# B&R Automation Studio project TD52 (part 132)

### module_SA.typ - Package data types
```iecst
TYPE
	tVIS2MM : 	STRUCT
		bPI_SelfTest : BOOL; (* Switch port injection to selftest *) (* OldName:bSAFIPITest; Cycle: *)
		bCanUpDevSel : ARRAY[0..12]OF BOOL; (* CAN updater device selection *) (* OldName:new PV; Cycle: *)
		bCanUpStart : BOOL; (* CAN updater start/stop button *) (* OldName:new PV; Cycle: *)
		iCanUpFwVersSel : INT; (* CAN updater firmware version selection *) (* OldName:new PV; Cycle: *)
		bSAFI_SL_Check : BOOL; (* SAFI safty loop testing button *) (* OldName:bSAFI_SL_Check; Cycle: *)
		bSAFI_ValveLashSet : ARRAY[0..24]OF BOOL; (*Valve lash adjusted*)
		bSAFI_ValveLashSetAll : BOOL; (*Valve lash adjusted all*)
		bCanUpDevSelAll : BOOL; (*Update all button*)
	END_STRUCT;
	tMM2VIS : 	STRUCT
		iCnt_SA_ComErr : ARRAY[0..12]OF DINT; (* SAFI communication error counter *) (* OldName:usSAFIComErrCnt; Cycle:  *)
		iTi_PI_DurationAvg : INT; (* port injection duration average *) (* OldName:usDurationAvg; Cycle: *)
		iTi_PI_DurationMax : INT; (* port injection duration maximum *) (* OldName:usDurationMax; Cycle: *)
		iTi_PI_DurationMin : INT; (* port injection duration minimum *) (* OldName:usDurationMin; Cycle: *)
		tSA_HW_Vers : ARRAY[0..12]OF _tSAFIHardwareINT; (* SAFI hardware version *) (* OldName:usSAFIHW; Cycle: *)
		rSA_SW_Vers : ARRAY[0..12]OF REAL; (* SAFI software version *) (* OldName:usSAFIVers; Cycle: *)
		rTi_SA_OpHours : ARRAY[0..12]OF REAL; (* SAFI operating hours *) (* OldName:ulSAFArbH; Cycle: *)
		iSA_SerialNr : ARRAY[0..12]OF DINT; (* SAFI serial number *) (* OldName:ulSAFSerNr; Cycle: *)
		tSA_ProdDate : ARRAY[0..12]OF _tSAFIProdDateINT; (* SAFI production date *) (* OldName:ulProdDate; Cycle: *)
		rT_SA_ElecTemp : ARRAY[0..12]OF REAL; (* SAFI electronic temperature *) (* OldName:ssSAFITemp; Cycle: *)
		iSA_ErrToothNr : ARRAY[0..12]OF INT; (* SAFI Error tooth number *) (* OldName:usErrZahnz; Cycle: *)
		rSA_FiltVers : ARRAY[0..12]OF REAL; (* SAFI KLS filter version *) (* OldName:usSAFFiltV; Cycle: *)
		bMsg3337 : BOOL; (* Message number 3337 *) (* OldName:bACamSign; Cycle: *)
		bMsg3335 : BOOL; (* Message number 3335 *) (* OldName:bAOverspeedErr; Cycle: *)
		bMsg3333 : BOOL; (* Message number 3333 *) (* OldName:bAParameter; Cycle: *)
		bMsg2256 : BOOL; (* Message number 2256 *) (* OldName:bAPICloseErr; Cycle: *)
		bMsg2253 : BOOL; (* Message number 2253 (prepared V4.05.00*) (* OldName:Port injetion duration error; Cycle: *)
		bMsg2254 : BOOL; (* Message number 2254 *) (* OldName:bAPIHardwareErr; Cycle: *)
		bMsg2255 : BOOL; (* Message number 2255 *) (* OldName:bAPIOpenErr; Cycle: *)
		bMsg2281 : BOOL; (* Message number 2281 *) (* OldName:bAPBCMemBurst; Cycle: *)
		bMsg3331 : BOOL; (* Message number 3331 *) (* OldName:bASAFIComErr; Cycle: *)
		bMsg3336 : BOOL; (* Message number 3336 *) (* OldName:bATriggerSign; Cycle: *)
		bMsg3330 : BOOL; (* Message number 3330 *) (* OldName:bASAFIHwErr; Cycle: *)
		bMsg3332 : BOOL; (* Message number 3332 *) (* OldName:bASAFIWrongVers; Cycle: *)
		bMsg3334 : BOOL; (* Message number 3334 *) (* OldName:bAIPDeviation; Cycle: *)
		bMsg3338 : BOOL; (* Message number 3338 *) (* OldName:bAOutputErr; Cycle: *)
		bMsg3343 : BOOL; (* Message number 3343 *) (* OldName:bAMORISErr; Cycle: *)
		bMsg3344 : BOOL; (* Message number 3344 *) (* OldName:bIgnPowerFail; Cycle: *)
		bMsg3345 : BOOL; (* Message number 3345 *) (* OldName:bSAFISafetyLoop; Cycle: *)
		bMsg3277 : BOOL; (* Message number 3277 *) (* OldName:bBCamSign; Cycle: *)
		bMsg3292 : BOOL; (* Message number 3292 *) (* OldName:bBCanErrRate; Cycle: *)
		bMsg3291 : BOOL; (* Message number 3291 *) (* OldName:bBConfigErr; Cycle: *)
		bMsg3293 : BOOL; (* Message number 3293 *) (* OldName:bBElectrTemp; Cycle: *)
		bMsg3294 : BOOL; (* Message number 3294 *) (* OldName:bBIgnPwrLim; Cycle: *)
		bMsg2824 : BOOL; (* not used at the moment!? *) (* OldName:bBIGNShutOff; Cycle: *)
		bMsg3288 : BOOL; (* Message number 3288 *) (* OldName:bBIgnVoltMax; Cycle: *)
		bMsg3287 : BOOL; (* Message number 3287 *) (* OldName:bBIgnVoltMin; Cycle: *)
		bMsg3286 : BOOL; (* Message number 3286 *) (* OldName:bBOffsetErr; Cycle: *)
		bMsg3278 : BOOL; (* Message number 3278 *) (* OldName:bBOutputErr; Cycle: *)
		bMsg3275 : BOOL; (* Message number 3275 *) (* OldName:bBOverspeedErr; Cycle: *)
		bMsg3273 : BOOL; (* Message number 3273 *) (* OldName:bBParameter; Cycle: *)
		bMsg2820 : BOOL; (* not used at the moment!? *) (* OldName:bBPICloseErr; Cycle: *)
		bMsg2818 : BOOL; (* not used at the moment!? *) (* OldName:bBPIHardwareErr; Cycle: *)
		bMsg2819 : BOOL; (* not used at the moment!? *) (* OldName:bBPIOpenErr; Cycle: *)
		bMsg2823 : BOOL; (* not used at the moment!? *) (* OldName:bBPIShutOff; Cycle: *)
		bMsg3271 : BOOL; (* Message number 3271 cylinder info value *) (* OldName:bBSAFIComErr; Cycle: *)
		bMsg3276 : BOOL; (* Message number 3276 cylinder info value *) (* OldName:bBTriggerSign; Cycle: *)
		bMsg3270 : BOOL; (* Message number 3270 cylinder info value *) (* OldName:bBSAFIHwErr; Cycle: *)
		bMsg3283 : BOOL; (* Message number 3283 cylinder info value *) (* OldName:bBMORISErr; Cycle: *)
		bMsg3284 : BOOL; (* Message number 3284 cylinder info value *) (* OldName:bBSAFIFwErr; Cycle: *)
		bMsg3272 : BOOL; (* Message number 3272 cylinder info value *) (* OldName:bBSAFIWrongVers; Cycle: *)
		bMsg3274 : BOOL; (* Message number 3274 cylinder info value *) (* OldName:bBIPDeviation; Cycle: *)
		bMsg2816 : BOOL; (* Message number 2816 cylinder info value *) (* OldName:bPIOpen; Cycle: *)
		bMsg2817 : BOOL; (* Message number 2817 cylinder info value *) (* OldName:bPIOpen; Cycle: *)
		bMsg3536 : BOOL; (* Message number 3536 cylinder info value *) (* OldName:bWCamSign; Cycle: *)
		bMsg3531 : BOOL; (* Message number 3531 cylinder info value *) (* OldName:bWCanErrRate; Cycle: *)
		bMsg3535 : BOOL; (* Message number 3535 cylinder info value *) (* OldName:bWConfigErr; Cycle: *)
		bMsg3539 : BOOL; (* Message number 3539 cylinder info value *) (* OldName:bWElectrTemp; Cycle: *)
		bMsg3551 : BOOL; (* Message number 3551 cylinder info value *) (* OldName:bWIgnPwrLim; Cycle: *)
		bMsg3549 : BOOL; (* Message number 3549 cylinder info value *) (* OldName:bWIgnVoltAvg; Cycle: *)
		bMsg3550 : BOOL; (* Message number 3550 cylinder info value *) (* OldName:bWIgnVoltDev; Cycle: *)
		bMsg3548 : BOOL; (* Message number 3548 cylinder info value *) (* OldName:bWIgnVoltMax; Cycle: *)
		bMsg3547 : BOOL; (* Message number 3547 cylinder info value *) (* OldName:bWIgnVoltMin; Cycle: *)
		bMsg3546 : BOOL; (* Message number 3546 cylinder info value *) (* OldName:bWOffsetErr; Cycle: *)
		bMsg3545 : BOOL; (* Message number 3545 cylinder info value *) (* OldName:bWOutputErr; Cycle: *)
		bMsg2585 : BOOL; (* Message number 2585 cylinder info value *) (* OldName:bWPIHardwareErr; Cycle: *)
		bMsg3530 : BOOL; (* Message number 3530 cylinder info value *) (* OldName:bWSAFIComErr; Cycle: *)
		bMsg3537 : BOOL; (* Message number 3537 cylinder info value *) (* OldName:bWTriggerSign; Cycle: *)
		bMsg3533 : BOOL; (* Message number 3533 cylinder info value *) (* OldName:bWSAFIFwErr; Cycle: *)
		bMsg3544 : BOOL; (* Message number 3544 cylinder info value *) (* OldName:bWMORISErr; Cycle: *)
		iMsg3277 : INT; (* Message number 3277 cylinder info value *) (* OldName:ucCamSign; Cycle: *)
		iMsg3275 : INT; (* Message number 3275 cylinder info value *) (* OldName:ucOverspeedErr; Cycle: *)
		iMsg3273 : INT; (* Message number 3273 cylinder info value *) (* OldName:ucParameter; Cycle: *)
		iMsg2820 : INT; (* Message number 2820 cylinder info value *) (* OldName:ucPICloseErr; Cycle: *)
		iMsg2819 : INT; (* Message number 2819 cylinder info value *) (* OldName:ucPIOpenErr; Cycle: *)
		iMsg3271 : INT; (* Message number 3271 cylinder info value *) (* OldName:ucSAFIComErr; Cycle: *)
		iMsg3276 : INT; (* Message number 3276 cylinder info value *) (* OldName:ucTriggerSign; Cycle: *)
		iMsg3270 : INT; (* Message number 3270 cylinder info value *) (* OldName:ucSAFIHwErr; Cycle: *)
		iMsg3272 : INT; (* Message number 3272 cylinder info value *) (* OldName:ucSAFIWrongVers; Cycle: *)
		iMsg3274 : INT; (* Message number 3274 cylinder info value *) (* OldName:ucIPDeviation; Cycle: *)
		iMsg3278 : INT; (* Message number 3278 cylinder info value *) (* OldName:ucOutputErr; Cycle: *)
		iMsg3283 : INT; (* Message number 3283 cylinder info value *) (* OldName:ucMORISErr; Cycle: *)
		iMsg3292 : INT; (* Message number 3292 cylinder info value *) (* OldName:ucCanErrRate; Cycle: *)
		iMsg3291 : INT; (* Message number 3291 cylinder info value *) (* OldName:ucConfigErr; Cycle: *)
		iMsg3293 : INT; (* Message number 3293 cylinder info value *) (* OldName:ucElectrTemp; Cycle: *)
		iMsg3294 : INT; (* Message number 3294 cylinder info value *) (* OldName:ucIgnPwrLim; Cycle: *)
		iMsg3288 : INT; (* Message number 3288 cylinder info value *) (* OldName:ucIgnVoltMax; Cycle: *)
		iMsg3287 : INT; (* Message number 3287 cylinder info value *) (* OldName:ucIgnVoltMin; Cycle: *)
		iMsg3286 : INT; (* Message number 3286 cylinder info value *) (* OldName:ucOffsetErr; Cycle: *)
		iMsg2818 : INT; (* Message number 2818 cylinder info value *) (* OldName:ucPIHardwareErr; Cycle: *)
		iMsg3284 : INT; (* Message number 3284 cylinder info value *) (* OldName:ucSAFIFwErr; Cycle: *)
		bMsg3532 : BOOL; (* not used at the moment!? *) (* OldName:SAFI wrong type of software; Cycle: *)
		bMsg3534 : BOOL; (* not used at the moment!? *) (* OldName:SAFI  parameter failure; Cycle: *)
		bMsg3538 : BOOL; (* not used at the moment!? *) (* OldName:SAFI hardware failure; Cycle: *)
		bMsg3543 : BOOL; (* not used at the moment!? *) (* OldName:Ignition point deviation too high; Cycle: *)
		bMsg3552 : BOOL; (* SAFI ignition power module overload *) (* OldName:Ignition power supply overload; Cycle: *)
		bMsg3553 : BOOL; (* Message number 3553 *) (* OldName:bWPBCConfNotOK; Cycle: *)
		bMsg3554 : BOOL; (* Message number 3554 *) (* OldName:bWPBCInvalidPar; Cycle: *)
		bMsg2214 : BOOL; (* Message number 2214 *) (* OldName:bAPBCSigErr; Cycle: *)
		bMsg2297 : BOOL; (* PI correct current control rate message *) (* OldName:new PV; Cycle: *)
		bMsg2800 : BOOL; (* PI correct current control warning message *) (* OldName:new PV; Cycle: *)
		bMsg2906 : BOOL; (* PI correct current control warning message *) (* OldName:new PV; Cycle: *)
		iMsg2906 : INT; (* PI correct current control warning message *) (* OldName:new PV; Cycle: *)
		bMsg2298 : BOOL; (* PI demagnetisation failure message *) (* OldName:new PV; Cycle: *)
		bMsg2907 : BOOL; (* PI demagnetisation failure message *) (* OldName:new PV; Cycle: *)
		iMsg2907 : INT; (* PI demagnetisation failure message *) (* OldName:new PV; Cycle: *)
		iSA_ERZuV : ARRAY[0..24]OF INT; (* Error Rate for spark delay  *) (* OldName:ucERZuV; Cycle: *)
		iSA_ERDurTol : ARRAY[0..24]OF INT; (* Error Rate for Duration Tolerance  *) (* OldName:ucERDurTol; Cycle: *)
		rCanUpProgress : REAL; (* CAN updater progress bar *) (* OldName:new PV; Cycle: *)
		rCanUpFwVers : ARRAY[0..5]OF REAL; (* CAN updater firmware versions *) (* OldName:new PV; Cycle: *)
		bSAFI2 : BOOL; (* CAN updater SAFI2 detected *) (* OldName:new PV; Cycle: *)
		iSA_PICurGrad : ARRAY[0..24]OF INT; (* port injection close current gradient *) (* OldName:new PV; Cycle: *)
		iSA_PICurGradAvg : INT; (* port injection close current gradient average *) (* OldName:new PV; Cycle: *)
		iSA_PICurGradMax : INT; (* port injection close current gradient maximum *) (* OldName:new PV; Cycle: *)
		iSA_PICurGradMin : INT; (* port injection close current gradient minimum *) (* OldName:new PV; Cycle: *)
		bMsg2299 : BOOL; (* alarm A2299 cylinder pressure saturation replaced with warning W9318 if RKS enabled *) (* OldName:new PV; Cycle: *)
		bMsg9318 : BOOL; (* W9318 Cylinder pressure sensor saturation *) (* OldName:new PV; Cycle: *)
		bMsg2898 : BOOL; (* Message number 2898 cylinder info value *) (* OldName:new PV; Cycle: *)
		iMsg2898 : INT; (* Message number 2818 cylinder info value *) (* OldName:new PV; Cycle: *)
		bMsg2910 : BOOL; (* Message number 2910 cylinder info value *) (* OldName:new PV; Cycle: *)
		iMsg2910 : INT; (* Message number 2910 MPM info value *) (* OldName:new PV; Cycle: *)
		iMsg3344 : INT; (* Message number 3344 MPM  info value *) (* OldName:new PV; Cycle: *)
		iCMSmain_SAFI_status : INT; (* SAFI Module Main CMS Status *)
		iCMSinit_SAFI_status : INT; (* SAFI Module CMS Init Status *)
		bMsg2476 : BOOL; (*Message number 2476 SPAx CAM deviation monitoring*)
		iU_SAFI_Win3 : ARRAY[0..24]OF UINT; (*Outlet valve closure noise*)
		iU_SAFI_Win3_Min : UINT; (*Outlet valve closure noise min*)
		iU_SAFI_Win3_Max : UINT; (*Outlet valve closure noise max*)
		iU_SAFI_Win3_Avg : UINT; (*Outlet valve closure noise average*)
		iU_SAFI_Win4 : ARRAY[0..24]OF UINT; (*Inlet valve closure noise*)
		iU_SAFI_Win4_Min : UINT; (*Inlet valve closure noise min*)
		iU_SAFI_Win4_Max : UINT; (*Inlet valve closure noise max*)
		iU_SAFI_Win4_Avg : UINT; (*Inlet valve closure noise average*)
		iCA_SAFI_Win3 : ARRAY[0..24]OF UINT; (*Outlet valve closure timing*)
		iCA_SAFI_Win3_Min : UINT; (*Outlet valve closure timing min*)
		iCA_SAFI_Win3_Max : UINT; (*Outlet valve closure timing max*)
		iCA_SAFI_Win3_Avg : UINT; (*Outlet valve closure timing average*)
		iCA_SAFI_Win4 : ARRAY[0..24]OF UINT; (*Inlet valve closure timing*)
		iCA_SAFI_Win4_Min : UINT; (*Inlet valve closure timing min*)
		iCA_SAFI_Win4_Max : UINT; (*Inlet valve closure timing max*)
		iCA_SAFI_Win4_Avg : UINT; (*Inlet valve closure timing average*)
		bMsg2334 : BOOL; (*Alarm 2334 Outlet valve closure noise high*)
		bMsg9027 : BOOL; (*Operating message 9027 Outlet valve closure noise high*)
		iMsg9027 : UINT; (*Operating message 9027 Outlet valve closure noise high - Cylinder info*)
		bMsg2335 : BOOL; (*Alarm 2335 Outlet valve closure noise high*)
		bMsg9028 : BOOL; (*Operating message 9028 Outlet valve closure noise high*)
		iMsg9028 : UINT; (*Operating message 9028 Outlet valve closure noise high - Cylinder info*)
		bSA_VCD_Active : BOOL; (*Enable visualization of VCD parameters for legacy versions*)
		bMsg9320 : BOOL; (*Warning 9320 Exhaust valve unbalance*)
		bMsg9045 : BOOL; (*Operating message 9045 Exhaust valve unbalance*)
		iMsg9045 : UINT; (*Operating message 9045 Exhaust valve unbalance - Cylinder info*)
		bMsg9321 : BOOL; (*Warning 9321 Intake valve unbalance*)
		bMsg9046 : BOOL; (*Operating message 9046 Intake valve unbalance*)
		iMsg9046 : UINT; (*Operating message 9046 Intake valve unbalance - Cylinder info*)
		bMsg2493 : BOOL; (*Warning 2493 - SAFI measurements frozen or alternating*)
		bMsg2939 : BOOL; (*Operating message 2939 - SAFI measurements frozen or alternating*)
		iMsg2939 : UINT; (*Operating message 2939 - SAFI measurements frozen or alternating - Cylinder info*)
		bP_Red_SAErr_Bar : BOOL; (*Bit to activate the SAFI power reduction bar in the HMI*)
		bMsg9066 : BOOL; (*Operating message 9066 Cylinder pressure sensor measuring signal failure*)
		iMsg9066 : UINT; (*Operating message 9066 Cylinder pressure sensor measuring signal failure - Cylinder info*)
		bMsg9350 : BOOL; (*W9350 - KLS21 ignition monitoring not available*)
		bMsg9050 : BOOL; (*B9050 - KLS21 ignition monitoring not available*)
		iMsg9050 : UINT; (*B9050 - KLS21 ignition monitoring not available - cylinder number*)
		iNum_SafiType : ARRAY[0..12]OF USINT; (*Type of device. Unknown: 0. SAFI1: 1. SAFI2 KLS: 2. SAFI2 DMR: 3. SAFI3: 4. KLS21: 5.*)
		iNum_SafiUpdBlock : USINT; (*Block the CAN update procedure*)
		bSAFI3 : BOOL; (*All installed devices are not SAFI1*)
	END_STRUCT;
	_tSAFISpeed : 	STRUCT
		InCan : UINT;
		In : UINT;
		ValOK : UINT;
		Time : UDINT;
	END_STRUCT;
	_tSAFIProdDateINT : 	STRUCT
		YYYY : INT;
		MM : INT;
		DD : INT;
	END_STRUCT;
	_tSAFIProdDate : 	STRUCT
		YYYY : UINT;
		MM : USINT;
		DD : USINT;
	END_STRUCT;
	_tSAFICurrPmmREAL : 	STRUCT
		Current : REAL;
		Time : REAL;
	END_STRUCT;
	_tSAFICurrPmm : 	STRUCT
		Current : USINT;
		Time : UINT;
	END_STRUCT;
	_tSAFICurr : 	STRUCT
		Current_Low : USINT;
		Current_High : USINT;
		Time_Low : UINT;
		Time_High : UINT;
	END_STRUCT;
	_SAFIError : 	STRUCT
		Error : ARRAY[0..5]OF USINT;
	END_STRUCT;
	_tSAFImdatas : 	STRUCT
		data1 : UINT;
		data2 : UINT;
		data3 : UINT;
	END_STRUCT;
	_tSAFImdatasExtend : 	STRUCT
		data1 : UINT;
		data2 : UINT;
		data3 : UINT;
		data4 : USINT;
	END_STRUCT;
	_tSAFIHardwareINT : 	STRUCT
		HW_OPTION : INT;
		HW_VERSION : INT;
	END_STRUCT;
	_tSAFIHardware : 	STRUCT
		HW_OPTION : USINT;
		HW_VERSION : USINT;
	END_STRUCT;
	tE_SAFI : 	STRUCT
		Error : ARRAY[0..1]OF USINT;
		pdata : ARRAY[0..41]OF USINT;
		runstop : ARRAY[0..2]OF USINT;
		smdata : ARRAY[0..9]OF USINT;
	END_STRUCT;
	_tEventSAFI : 	STRUCT
		conf : ARRAY[0..35]OF USINT;
		zuend : ARRAY[0..1]OF USINT;
		error : USINT;
		sdata : ARRAY[0..4]OF USINT;
		idata : ARRAY[0..30]OF USINT;
		kdata : ARRAY[0..30]OF USINT;
		ddata : ARRAY[0..53]OF USINT;
		dmdata1 : ARRAY[0..5]OF USINT;
		kmdata : ARRAY[0..7]OF USINT;
		dmdata2 : ARRAY[0..15]OF USINT;
		smdata : ARRAY[0..9]OF USINT;
		status : ARRAY[0..11]OF USINT;
		bez : USINT;
		ref : USINT;
		cur : USINT;
		diag : ARRAY[0..18]OF USINT;
	END_STRUCT;
	tPIcurrentREAL : 	STRUCT
		current : REAL;
		duration : REAL;
	END_STRUCT;
	tPIrecoveryREAL : 	STRUCT
		delay : REAL;
		current : REAL;
		duration : REAL;
	END_STRUCT;
	tPIpulldet1REAL : 	STRUCT
		level : REAL;
		st_time : REAL;
	END_STRUCT;
	tPIopdet1REAL : 	STRUCT
		st_time : REAL;
		duration : REAL;
	END_STRUCT;
	tPIopdet2REAL : 	STRUCT
		grad_ul : REAL;
		grad_ll : REAL;
		rate : REAL;
	END_STRUCT;
	tPIclosdet1REAL : 	STRUCT
		set_current : REAL;
		set_duration : REAL;
	END_STRUCT;
	tPIclosdet2REAL : 	STRUCT
		duration : REAL;
		grad_curr : REAL;
		grad_curr_var : REAL;
	END_STRUCT;
	tPIaverageREAL : 	STRUCT
		average_MUX_6_7 : REAL;
		average_MUX_8_9 : REAL;
	END_STRUCT;
	CanDeviceGo : 	STRUCT
		CANDevGo : ARRAY[0..1]OF USINT;
		ECANDevGo : USINT;
	END_STRUCT;
	_tMonicLimitREAL : 	STRUCT
		limit : REAL;
		kind : REAL;
		delay : REAL;
	END_STRUCT;
	_tMonicLimit : 	STRUCT
		limit : USINT;
		kind : USINT;
		delay : USINT;
	END_STRUCT;
	IN_SA_struct : 	STRUCT
		iIdx_OMSS : INT; (* operationg mode selection switch *) (* OldName:BWS_HA; Cycle:5 *)
		iIdx_OMSS_TC2 : INT; (* operationg mode selection switch *) (* OldName:BWS_HA; Cycle:5 *)
		bEng_Dem_TC2 : BOOL; (* module demanded *) (* OldName:M_AGFD; Cycle:2 *)
		bEng_Dem : BOOL; (* module demanded *) (* OldName:M_AGFD; Cycle:5 *)
		iSt_OpMode : UDINT; (* engine operation mode *) (* OldName:StopM; Cycle:5 *)
		rCA_Ign_Act : ARRAY[0..24]OF REAL; (* actual cylinder ignition point *) (* OldName:ZZPCyl ; Cycle:2 *)
		bIgn_Dem_TC1 : BOOL; (* demand ignition *) (* OldName:ZUEND; Cycle:1 *)
		bIgn_Dem_TC2 : BOOL; (* demand ignition *) (* OldName:ZUEND; Cycle:2 *)
		bIgn_Dem : BOOL; (* demand ignition *) (* OldName:ZUEND; Cycle:5 *)
		bGV_On : BOOL; (* command open gas valves *) (* OldName:M_GASV; Cycle:2 *)
		tPIopenH : ARRAY[0..12]OF tPIopen; (* PI open point and open duration for high cylinder *) (* OldName:SAFI.tPI.tPIopenH; Cycle:2 *)
		tPIopenL : ARRAY[0..12]OF tPIopen; (* PI open point and open duration for low cylinder *) (* OldName:SAFI.tPI.tPIopenL; Cycle:2 *)
		bEng_Start_TC2 : BOOL; (*engine start*) (*OldName:M_STRT; Cycle:5*)
		bEng_Start : BOOL; (*engine start*) (*OldName:M_STRT; Cycle:5*)
		bIgn_SelfTest : BOOL; (* Switch ignition system to selftest  *) (* OldName:GoSelftest; Cycle:5 *)
		tAB2SA_TC2 : AmmBase2MM; (* AMM base to SAFI data transfer *) (* OldName:QUITT_WA; Cycle:2 *)
		tAB2SA : AmmBase2MM; (* AMM base to SAFI data transfer *) (* OldName:QUITT_WA; Cycle:5 *)
		iCANIdent : UDINT; (* CAN identifier from HalIO *) (* OldName:new PV; Cycle:7 *)
		iCANIdent_TC8 : UDINT; (* CAN identifier from HalIO *) (* OldName:new PV; Cycle:8 *)
		iCANIdentIGN2 : UDINT; (* CAN identifier of the 2nd CAN card from HalIO *) (* OldName:new PV; Cycle:8 *)
		iCANIdentIGN2_TC8 : UDINT; (* CAN identifier of the 2nd CAN card from HalIO *) (* OldName:new PV; Cycle:8 *)
		iMisfCyl : UDINT; (* cylinder misfire parameter *) (* OldName:MissfCyl; Cycle:2 *)
		iMisfCyl_TC2 : UDINT; (* cylinder misfire parameter *) (* OldName:MissfCyl; Cycle:2 *)
		tPB2MM : ParaBase2MM_type; (* Data exchange structure to ParaBase *) (* OldName:new PV; Cycle:5 *)
		tMO_PwrReply_TC5 : HALioDi_Type; (* DI: MORIS Ignition Power Module On *) (* OldName:DI_IgnPwrReply; Cycle:2 *)
		tMO_PwrReply : HALioDi_Type; (* DI: MORIS Ignition Power Module On *) (* OldName:DI_IgnPwrReply; Cycle:5 *)
		tMO_PwrReply2 : HALioDi_Type; (* DI: MORIS Ignition Power Module On *) (* OldName:new PV; Cycle:5 *)
		tMO_PwrReply3 : HALioDi_Type; (* DI: MORIS Ignition Power Module On *) (* OldName:new PV; Cycle:5 *)
		tMO_PwrReply4 : HALioDi_Type; (* DI: MORIS Ignition Power Module On *) (* OldName:new PV; Cycle:5 *)
		tMO_SaftyLoop_TC2 : HALioDi_Type; (* DI: MORIS Savety loop closed *) (* OldName:DI_MO_SL_OK; Cycle:2 *)
		tMO_SaftyLoop : HALioDi_Type; (* DI: MORIS Savety loop closed *) (* OldName:DI_MO_SL_OK; Cycle:5 *)
		tSafetyLoop_Eng_TC2 : HALioDi_Type; (* DI: Safety Loop closed *) (* OldName:RUHE; Cycle:2 *)
		tSafetyLoop_Eng : HALioDi_Type; (* DI: Safety Loop closed *) (* OldName:RUHE; Cycle:5 *)
		tMO_PowerOverload : HALioDi_Type; (* DI: SAFI ignition power module overload *) (* OldName:DI_IgnPowerOverload; Cycle:5 *)
		tMO_PowerOverload2 : HALioDi_Type; (* DI: SAFI ignition power module overload *) (* OldName:new PV; Cycle:5 *)
		tMO_PowerOverload3 : HALioDi_Type; (* DI: SAFI ignition power module overload *) (* OldName:new PV; Cycle:5 *)
		tMO_PowerOverload4 : HALioDi_Type; (* DI: SAFI ignition power module overload *) (* OldName:new PV; Cycle:5 *)
		tSafetyLoop_EmStop : HALioDi_Type; (* DI safety loop - emergency stop *) (* OldName:DI_SIS; Cycle:5 *)
		tGCB_On : HALioDi_Type; (*DI: generator circuit breaker closed *) (*OldName:GCB_ON; Cycle:2;*)
		tGCB_On_TC5 : HALioDi_Type; (*DI: generator circuit breaker closed *) (*OldName:GCB_ON; Cycle:2;*)
		iECanDevGo : USINT; (* event status CAN device go *) (* OldName:new PV; Cycle:2 *)
		bSimWinMOD_Active : BOOL; (* WinMode simulation active *) (* OldName:new PV; Cycle:2*)
		rP_Act_Norm_Filt : REAL; (* actual power related to rP_Nom filtered T=1s *) (*OldName:P_IST; Cycle:2*)
		rP_Act_Norm_Filt_TC5 : REAL; (* actual power related to rP_Nom filtered T=1s *) (*OldName:P_IST; Cycle:5*)
		iIdx_Gtyp_Dem : INT; (* actual gassort 1..4 *) (* OldName: gasart; Cycle:5; *)
		bLimpHomeCyl : ARRAY[0..24]OF BOOL; (* limp home if PBC in-cylinder pressure sensor failure *) (* OldName: bLimpHomeCyl; Cycle:2; *)
		bCUp_Man : ARRAY[0..24]OF BOOL; (* SAFI curve upload manuel selection *) (* OldName: ManualUpload; Cycle:2; *)
		rLam_Eng_LL_Set : REAL; (* Leanox Lambda set point *) (* OldName: ssPosGasmixerNominal; Cycle:2; *)
		rPr_Ch_P2s_Avg_TC2 : REAL; (* actual charge pressure before throttle valve (P2s) *) (* OldName: new PV; Cycle:2; *)
		rPr_Ch_P2s_Avg : REAL; (* actual charge pressure before throttle valve (P2s) *) (* OldName: new PV; Cycle:5; *)
		rT_Ch_T2s_Avg_TC2 : REAL; (* actual charge temperature (T2s) *) (* OldName: new PV; Cycle:2; *)
		rT_Ch_T2s_Avg : REAL; (* actual charge temperature (T2s) *) (* OldName: new PV; Cycle:5; *)
		bTrip_IPC_MSF : BOOL; (* Trip: A2214 Cylinder pressure sensor measuring signal failure Prio2*) (* OldName: bAKnockSigErr_DMR; Cycle:5; *)
		STP_STRT : BOOL; (*  tooth to tooth --> air starter off *) (* OldName: new PV; Cycle:5; *) (*V04.04.00.00*)
		bGridCode_ON : BOOL; (*any dyn. GridCode function activated*)
		bFastStart_ready_running : BOOL; (*Engine ready for fast start (engine stopped) OR fast start in action (until target load reached for the first time) *)
		bCANCntReset : BOOL; (* CAN error counter value reset *) (*OldName: bCANCounterReset; Cycle:5;*)
		tSPAx_CamDev : HALioDi_Type; (*DI: SPAx CAM deviation monitoring*) (* OldName: new PV; Cycle:5; *)
		bP_Red_SAErr : BOOL; (*Trigger SAFI power reduction*)
		bIC_IgnEngergy_Hi : BOOL; (*IC Warning Maximum Energy Exceeded*)
	END_STRUCT;
	OUT_SA_struct : 	STRUCT
		rN_IgnSAFI_Act : REAL; (* Engine speed measured by ignition SAFI *) (* OldName:ZDGSpeed; Cycle:2 *)
		bIgnOperating : BOOL; (* Ignition in Operation *) (* OldName:ZIB; Cycle:2 *)
		rT_EG_Cyl : ARRAY[0..24]OF REAL; (* cylinder exhaust gas temperatures *) (* OldName:t_zyl; Cycle:5 *)
		iU_SAFI_Win1 : ARRAY[0..24]OF INT; (* cylinder values of KLS window 1 *) (* OldName:Fenst1; Cycle:5 *)
		iU_SAFI_Win2 : ARRAY[0..24]OF INT; (* cylinder values of KLS window 2 *) (* OldName:Fenst2; Cycle:5 *)
		iU_SAFI_Win3 : ARRAY[0..24]OF INT; (* cylinder values of KLS window 3 *) (* OldName:Fenst3; Cycle:5 *)
		iU_SAFI_Win4 : ARRAY[0..24]OF INT; (* cylinder values of KLS window 4 *) (* OldName:Fenst4; Cycle:5 *)
		tMS_PBC0 : ARRAY[0..12]OF _tSAFImdatas; (* Pressure based control measuring data 0 *) (* OldName:DMR_md0; Cycle:5 *)
		tMS_PBC1 : ARRAY[0..12]OF _tSAFImdatas; (* Pressure based control measuring data 1 *) (* OldName:DMR_md1; Cycle:5 *)
		tMS_PBC2 : ARRAY[0..12]OF _tSAFImdatas; (* Pressure based control measuring data 2 *) (* OldName:DMR_md2; Cycle:5 *)
		tMS_PBC3 : ARRAY[0..12]OF _tSAFImdatas; (* Pressure based control measuring data 3 *) (* OldName:DMR_md3; Cycle:5 *)
		tMS_PBC4 : ARRAY[0..12]OF _tSAFImdatas; (* Pressure based control measuring data 4 *) (* OldName:DMR_md4; Cycle:5 *)
		tMS_PBC5 : ARRAY[0..12]OF _tSAFImdatas; (* Pressure based control measuring data 5 *) (* OldName:DMR_md5; Cycle:5 *)
		tMS_PBC6 : ARRAY[0..12]OF _tSAFImdatas; (* Pressure based control measuring data 6 *) (* OldName:DMR_md6; Cycle:5 *)
		tMS_PBC7 : ARRAY[0..12]OF _tSAFImdatas; (* Pressure based control measuring data 7 *) (* OldName:DMR_md7; Cycle:5 *)
		tMS_PBC8 : ARRAY[0..12]OF _tSAFImdatas; (* Pressure based control measuring data 8 *) (* OldName:DMR_md8; Cycle:5 *)
		tMS_PBC9 : ARRAY[0..12]OF _tSAFImdatas; (* Pressure based control measuring data 9 *) (* OldName:DMR_md9; Cycle:5 *)
		tMS_PBC10 : ARRAY[0..12]OF _tSAFImdatas; (* Pressure based control measuring data 10 *) (* OldName:DMR_md10; Cycle:5 *)
		tMS_PBC11 : ARRAY[0..12]OF _tSAFImdatas; (* Pressure based control measuring data 11 *) (* OldName:DMR_md11; Cycle:5 *)
		tMS_PBC12 : ARRAY[0..12]OF _tSAFImdatas; (* Pressure based control measuring data 12 *) (* OldName:DMR_md12; Cycle:5 *)
		tMS_PBC13 : ARRAY[0..12]OF _tSAFImdatas; (* Pressure based control measuring data 13 *) (* OldName:DMR_md13; Cycle:5 *)
		tMS_PBC14 : ARRAY[0..12]OF _tSAFImdatas; (* Pressure based control measuring data 14 *) (* OldName:DMR_md14; Cycle:5 *)
		tMS_PBC15 : ARRAY[0..12]OF _tSAFImdatas; (* Pressure based control measuring data 15 *) (* OldName:DMR_md15; Cycle:5 *)
		tMS_PBC16 : ARRAY[0..12]OF _tSAFImdatas; (* Pressure based control measuring data 16 *) (* OldName:DMR_md16; Cycle:5 *)
		tMS_PBC17 : ARRAY[0..12]OF _tSAFImdatas; (* Pressure based control measuring data 17 *) (* OldName:DMR_md17; Cycle:5 *)
		tMS_PBC18 : ARRAY[0..12]OF _tSAFImdatas; (* Pressure based control measuring data 18 *) (* OldName:DMR_md18; Cycle:5 *)
		tMS_PBC19 : ARRAY[0..12]OF _tSAFImdatas; (* Pressure based control measuring data 19 *) (* OldName:DMR_md19; Cycle:5 *)
		tMS_PBC20 : ARRAY[0..12]OF _tSAFImdatasExtend; (* Pressure based control measuring data 20*)
		tMS_PBC21 : ARRAY[0..12]OF _tSAFImdatasExtend; (* Pressure based control measuring data 21*)
		b_IgnSAFI_SelfTestBack : BOOL; (* Feedback: Ignition system SAFI is in selftest mode *) (* OldName:bSAFISelfTest; Cycle:5 *)
		rU_IgnSAFI_Max : REAL; (* maximum ignition voltage  *) (* OldName:MaxVolt; Cycle:5 *)
		rU_IgnSAFI_Min : REAL; (* minimum ignition voltage  *) (* OldName:MinVolt; Cycle:5 *)
		rU_IgnSAFI_Cyl : ARRAY[0..24]OF REAL; (* ignition voltage for each cylinder  *) (* OldName:V_Zyl; Cycle:5 *)
		rU_IgnSAFI_Avg : REAL; (* ignition voltage average *) (* OldName:AvgVolt; Cycle:5 *)
		tSAFI_CanGo : CanDeviceGo; (* Start / Stop CAN communication *) (* OldName:CANDevGo; Cycle:5 *)
		rN_IgnSAFI_LastValOK : REAL; (* last sent speed value from one of the SAFI devices *) (* OldName:n_lastValOK; Cycle:2 *)
		tSA2AB : MM2AmmBase; (* SAFI module to AMM base data transfer *) (* OldName:new PV; Cycle:2 *)
		tSA2PB : MM2ParaBase_type; (* Data exchange structure to ParaBase *) (* OldName:new PV; Cycle:5 *)
		tMO_PwrRequest : HALioDo_Type; (* DO: MORIS Ignition Power Module Request *) (* OldName:DO_IgnPwrRequest; Cycle:5 *)
		tMO_PwrRequest2 : HALioDo_Type; (* DO: MORIS Ignition Power Module Request *) (* OldName:new PV; Cycle:5 *)
		tMO_PwrRequest3 : HALioDo_Type; (* DO: MORIS Ignition Power Module Request *) (* OldName:new PV; Cycle:5 *)
		tMO_PwrRequest4 : HALioDo_Type; (* DO: MORIS Ignition Power Module Request *) (* OldName:new PV; Cycle:5 *)
		bPBCSensErr : ARRAY[0..24]OF BOOL; (* error info for PBC *) (* OldName:bZM_PBCSensErr; Cycle:5 *)
		bPBCCompLineCheck : ARRAY[0..24]OF BOOL; (* error info for PBC *) (* OldName:bPBCCompLineCheck; Cycle:5 *)
		bPBCNegVoltCheck : ARRAY[0..24]OF BOOL; (* error info for PBC *) (* OldName:bPBCNegVoltCheck; Cycle:5 *)
		bPBCNegPresCheck : ARRAY[0..24]OF BOOL; (* error info for PBC *) (* OldName:bPBCNegPresCheck; Cycle:5 *)
		bPBCPresSlopeCheck : ARRAY[0..24]OF BOOL; (* error info for PBC *) (* OldName:bPBCPresSlopeCheck; Cycle:5 *)
		bPBCSlowDriftCheck : ARRAY[0..24]OF BOOL; (* error info for PBC *) (* OldName:bPBCSlowDriftCheck; Cycle:5 *)
		bPBCConfNotOK : ARRAY[0..12]OF BOOL; (* error info for PBC *) (* OldName:bPBCConfNotOK; Cycle:5 *)
		bPBCMemBurst : ARRAY[0..24]OF BOOL; (* error info for PBC *) (* OldName:bPBCMemBurst; Cycle:5 *)
		bSAFIPBCConfNotOK : BOOL; (* blocking of start because SAFI PBC parameter are not valid *) (* OldName:bSAFIPBCConfNotOK; Cycle:2 *)
		tCUp : ARRAY[0..24]OF tCup_Perm; (* SAFI curve upload data *) (* OldName:tCup; Cycle:2 *)
		iCUpStack : ARRAY[0..23]OF USINT; (* SAFI curve upload stack *) (* OldName:Stack; Cycle:2 *)
		bPBCInvalidPar : ARRAY[0..12]OF BOOL; (* SAFI invalid PBC parameter *) (* OldName:bPBCInvalidPar; Cycle:2 *)
		rSA_SW_Vers : ARRAY[0..12]OF REAL; (* SAFI software version *) (* OldName:usSAFIVers; Cycle: *)
		rSA_FiltVers : ARRAY[0..12]OF REAL; (* SAFI KLS filter version *) (* OldName:usSAFFiltV; Cycle: *)
		rT_SA_ElecTemp : ARRAY[0..12]OF REAL; (* SAFI electronic temperature *) (* OldName:ssSAFITemp; Cycle: *)
		rSA_PBC_Sens : ARRAY[0..12]OF REAL; (* PBC sensor sensitivity [mV/bar] *) (* new PV; Cycle: 2*)
		bPBCCPSSat : ARRAY[0..24]OF BOOL; (* Cylinder pressure sensor saturation flag for cyl X *) (* new PV; Cycle: 2*)
		tE_SAFI : ARRAY[0..12]OF _tEventSAFI; (* SAFI CAN Events *)
		iCnt_SA_ComErr : ARRAY[0..12]OF DINT; (* SAFI communication error counter *) (* OldName:usSAFIComErrCnt; Cycle:  *)
		iSA_ERZuV : ARRAY[0..24]OF INT; (* Error Rate for spark delay  *) (* OldName:ucERZuV; Cycle: *)
		iSA_ERDurTol : ARRAY[0..24]OF INT; (* Error Rate for Duration Tolerance  *) (* OldName:ucERDurTol; Cycle: *)
		bSA_PBCFrozenAltern : ARRAY[0..24]OF BOOL; (*DMR knock signal or IMEP frozen or alternating*)
		bSA_Win1FrozenAltern : ARRAY[0..24]OF BOOL; (*Knock noise signal frozen or alternating*)
		iT_EG_CylFault : ARRAY[0..24]OF UINT; (*0 = No fault / bit0 = SAFI re-para active / bit1 = Exhaust gas temperature signal frozen or alternating*)
		rP_Red_SAErr_Norm : REAL; (* Power reduction by CAN communication failure for half or more SAFI or too many SAFI reboots*)
		bSA_CfgDone : BOOL; (*All SAFI in operation mode*)
		rIHR : ARRAY[0..24]OF REAL; (*Integrated heat release [kJ/m2]*)
		rU_Ign_Max_LimHi : REAL; (* Maximum ignition voltage high limit *)
		bMsg9318_Set : BOOL; (* W9318 cylinder pressure sensor saturation is set *)
	END_STRUCT;
	tPIclosgrad : 	STRUCT
		PICurGrad : INT;
		PCICurGrad : INT;
	END_STRUCT;
	tPIMode : 	STRUCT
		EnabRun : BOOL;
		PIself : BOOL;
		PCIself : BOOL;
		PIclose : BOOL;
		PCIclose : BOOL;
		MAct_6_7 : BOOL;
		MAct_8_9 : BOOL;
		Bit08 : BOOL;
		Bit09 : BOOL;
		Bit10 : BOOL;
		Bit11 : BOOL;
		Bit12 : BOOL;
		Bit13 : BOOL;
		Bit14 : BOOL;
		Bit15 : BOOL;
		Bit16 : BOOL;
	END_STRUCT;
	tPIopen : 	STRUCT
		timing : UINT;
		duration : UINT;
	END_STRUCT;
	tPIcurrent : 	STRUCT
		current : USINT;
		duration : UINT;
	END_STRUCT;
	tPIrecovery : 	STRUCT
		delay : UINT;
		current : SINT;
		duration : UINT;
	END_STRUCT;
	tPIaverage : 	STRUCT
		average_MUX_6_7 : USINT;
		average_MUX_8_9 : USINT;
	END_STRUCT;
	tPICurGrad : 	STRUCT
		ssFiFo : ARRAY[0..10]OF INT;
		slSum : DINT;
		ssAvg : INT;
	END_STRUCT;
	tPI : 	STRUCT
		Mode : UINT;
		tPIopenH : tPIopen;
		tPIopenL : tPIopen;
		tPIcurr1 : tPIcurrent;
		tPIcurr2 : tPIcurrent;
		tPIcurr3 : tPIcurrent;
		PIcurr4 : USINT;
		tPIrecov : tPIrecovery;
		tPIpudet1 : tPIpulldet1;
		tPIpudet2 : tPIpulldet2;
		tPIpudet3 : tPIpulldet3;
		tPIopdet1 : tPIopdet1;
		tPIopdet2 : tPIopdet2;
		tPIopdet3 : tPIopdet3;
		tPIopdet4 : tPIopdet4;
		PIclotim : UINT;
		tPIclodet0 : tPIclosdet0;
		tPIclodet1 : tPIclosdet1;
		tPIclodet2 : tPIclosdet2;
		tPIclodet3 : tPIclosdet3;
		tPIclodet4 : tPIclosdet4;
		tPIclodet5 : tPIclosdet5;
		tPCopenH : tPCopen;
		tPCopenL : tPCopen;
		tPCcurr1 : tPCcurrent;
		tPCcurr2 : tPCcurrent;
		tPCcurr3 : tPCcurrent;
		PCcurr4 : USINT;
		tPCrecov : tPCrecovery;
		tPCpudet1 : tPCpulldet1;
		tPCpudet2 : tPCpulldet2;
		tPCopdet1 : tPCopdet1;
		tPCopdet2 : tPCopdet2;
		tPCopdet3 : tPCopdet3;
		tPCfree : tPCfree;
		PCclodet1 : UINT;
		tPCclodet2 : tPCclosdet2;
		tPCclodet3 : tPCclosdet3;
		ShOffRate : USINT;
		tAverage : tPIaverage;
		tPIdemagL : tPIdemag;
		tPIdemagH : tPIdemag;
		tPIcurrCtrL : tPIcurrCtrL;
		tPIcurrCtrH : tPIcurrCtrH;
		ucValveON : USINT;
		tVaOpenL : _tSAFImdatas;
		tVaOpenH : _tSAFImdatas;
		tCurrGradL : tPIclosgrad;
		tCurrGradH : tPIclosgrad;
	END_STRUCT;
	tSAFI : 	STRUCT
		tPI : tPI;
		tError : ARRAY[0..1]OF _SAFIError;
		E_SAFI : tE_SAFI;
	END_STRUCT;
	tPIpulldet1 : 	STRUCT
		level_L : UINT;
		level_H : UINT;
	END_STRUCT;
	tPIpulldet2 : 	STRUCT
		st_time_L : UINT;
		st_time_H : UINT;
	END_STRUCT;
	tPIpulldet3 : 	STRUCT
		duration_L : UINT;
		duration_H : UINT;
		rate : USINT;
	END_STRUCT;
	tPIopdet1 : 	STRUCT
		st_time_L : UINT;
		st_time_H : UINT;
	END_STRUCT;
	tPIopdet2 : 	STRUCT
		duration_L : UINT;
		duration_H : UINT;
	END_STRUCT;
	tPIopdet3 : 	STRUCT
		up_level_L : UINT;
		up_level_H : UINT;
	END_STRUCT;
	tPIopdet4 : 	STRUCT
		lo_level_L : UINT;
		lo_level_H : UINT;
		rate : USINT;
	END_STRUCT;
	tPIclosdet0 : 	STRUCT
		FailR_L : UINT;
		FailR_H : UINT;
	END_STRUCT;
	tPIclosdet1 : 	STRUCT
		st_time_L : UINT;
		st_time_H : UINT;
	END_STRUCT;
	tPIclosdet2 : 	STRUCT
		set_current_L : USINT;
		set_current_H : USINT;
	END_STRUCT;
	tPIclosdet3 : 	STRUCT
		set_duration_L : UINT;
		set_duration_H : UINT;
	END_STRUCT;
	tPIclosdet4 : 	STRUCT
		duration_L : UINT;
		duration_H : UINT;
		cur_gradient_L : INT;
	END_STRUCT;
	tPIclosdet5 : 	STRUCT
		cur_gradient_H : INT;
		var_limit_L : UINT;
		var_limit_H : UINT;
	END_STRUCT;
	tPCopen : 	STRUCT
		timing : UINT;
		duration : UINT;
	END_STRUCT;
	tPCcurrent : 	STRUCT
		current : USINT;
		duration : UINT;
	END_STRUCT;
	tPCrecovery : 	STRUCT
		delay : UINT;
		current : SINT;
		duration : UINT;
	END_STRUCT;
	tPCpulldet1 : 	STRUCT
		level : UINT;
		st_time : UINT;
	END_STRUCT;
	tPCpulldet2 : 	STRUCT
		duration : UINT;
		current : UINT;
		rate : USINT;
	END_STRUCT;
	tPCopdet1 : 	STRUCT
		st_time : UINT;
		duration : UINT;
	END_STRUCT;
	tPCopdet2 : 	STRUCT
		upper_lvl : UINT;
		lower_lvl : UINT;
		rate : USINT;
	END_STRUCT;
	tPCopdet3 : 	STRUCT
		min_curr : UINT;
		rate : USINT;
	END_STRUCT;
	tPCfree : 	STRUCT
		free : UINT;
	END_STRUCT;
	tPCclosdet2 : 	STRUCT
		set_current : USINT;
		set_duration : UINT;
	END_STRUCT;
	tPCclosdet3 : 	STRUCT
		duration : UINT;
		grad_curr : INT;
		grad_curr_var : UINT;
	END_STRUCT;
	tDMR_ref : 	STRUCT
		boost_pr : INT;
		mix_temp : INT;
	END_STRUCT;
	Pressure : 	STRUCT
		Low : ARRAY[0..719]OF UINT;
		LowCA : ARRAY[0..719]OF UINT;
		High : ARRAY[0..719]OF UINT;
		HighCA : ARRAY[0..719]OF UINT;
	END_STRUCT;
	tCup_Pm : 	STRUCT
		Perm : ARRAY[0..24]OF tCup_Perm;
	END_STRUCT;
	tCup_Perm : 	STRUCT
		Press : ARRAY[0..719]OF UINT;
		day : UINT;
		month : UINT;
		year : UINT;
		hour : UINT;
		minute : UINT;
		millisec : UDINT;
		rLam_Eng_LL_Set : REAL;
		rPr_Eng_P2s : REAL;
		rT_Eng_T2s : REAL;
		rP_Act_Norm_Filt : REAL;
	END_STRUCT;
	rtctime_typ : 	STRUCT
		year : UINT;
		month : USINT;
		day : USINT;
		reserve : USINT;
		hour : USINT;
		minute : USINT;
		second : USINT;
		millisec : UINT;
		microsec : UINT;
	END_STRUCT;
	tPIdemag : 	STRUCT
		delay : UINT;
		duration : UINT;
		up_limit : USINT;
	END_STRUCT;
	tPIcurrCtrL : 	STRUCT
		delay : UINT;
		duration : UINT;
		level : USINT;
	END_STRUCT;
	tPIcurrCtrH : 	STRUCT
		delay : UINT;
		duration : UINT;
		level : USINT;
		rate : USINT;
	END_STRUCT;
	tDiag : 	STRUCT
		ParaFail : tParaFail;
	END_STRUCT;
	tParaFail : 	STRUCT
		Id : UINT;
		Mux : USINT;
		Nr : USINT;
	END_STRUCT;
END_TYPE
```

### Module_SAPara.typ - Package data types
```iecst
TYPE
	PROGRAMMER_INFO : 	STRUCT
		DO_NOT_SORT_PARA : STRING[40] := 'DO NOT CHANGE PARAMETER SORTING!'; (*DO NOT CHANGE PARAMETER SORTING!*) (*ADD NEW PARAMETER ONLY AT THE END OF THE Para STRUCTURE. DO NOT DELETE existing Para items.*)
	END_STRUCT;
	Para_SA_struct : 	STRUCT
		rCA_AdvTimeLim : REAL; (*PARA [12065]: advanced ingnition timing 1/10 deg *) (* OldName:AdvTimLi; Cycle: *)
		bSA_PI_CloDetActive : BOOL; (*PARA [12121]: TRUE = SAFI PI close detection is enabled/active *) (* OldName:bCloDet_Act; Cycle: *)
		bSA_Active : BOOL; (*PARA [12114]: TRUE = SAFI is enabled/active *) (* OldName:bSAFI_Act; Cycle: *)
		bSA_PBC_Active : BOOL; (*PARA [12119]: TRUE = SAFI PBC function is enabled/active *) (* OldName:bSAFIDMR_Act; Cycle: *)
		bSA_EG_Active : BOOL; (*PARA [12115]: TRUE = SAFI exh. temp. measur. is enabled/active *) (* OldName:bSAFIExhT_Act; Cycle: *)
		bSA_HV_Active : BOOL; (*PARA [12116]: TRUE = SAFI high volt. measur. is enabled/active *) (* OldName:bSAFIHS_Act; Cycle: *)
		bSA_Ign_Active : BOOL; (*PARA [12117]: TRUE = SAFI ignition function is enabled/active *) (* OldName:bSAFIIgn_Act; Cycle: *)
		bSA_KLS_Active : BOOL; (*PARA [12118]: TRUE = SAFI KLS function is enabled/active *) (* OldName:bSAFIKLS_Act; Cycle: *)
		bSA_PI_Active : BOOL; (*PARA [12120]: TRUE = SAFI port injection is enabled/active *) (* OldName:bSAFIPI_Act; Cycle: *)
		rN_EngNom : REAL; (*PARA [12128]: engine nominal speed *) (* OldName:n_nenn; Cycle: *)
		rN_OvrSpeed : REAL; (*PARA [12129]: Ignition overspeed limit *) (* OldName:OvrSpeed; Cycle: *)
		rCA_RetTimeLim : REAL; (*PARA [12066]: Retard ignition timing limit 1/10 deg  *) (* OldName:RetTimLi; Cycle: *)
		rSA_PI_opdet2_rate : REAL; (*PARA [12145]: SAFI PI opdet2_rate *) (* OldName:SAFI_tPI_tPIopdet2_ratePMM; Cycle: *)
		rSA_PI_pudet2_rate : REAL; (*PARA [12146]: SAFI PI pudet2_rate *) (* OldName:SAFI_tPI_tPIpudet2_ratePMM; Cycle: *)
		tSA_Ign_0 : _tSAFICurrPmmREAL; (* Para: SAFI ignition current / duration setting 0 *) (* OldName:SAFICurr0PMM; Cycle: *)
		tSA_Ign_1 : _tSAFICurrPmmREAL; (* Para: SAFI ignition current / duration setting 1 *) (* OldName:SAFICurr1PMM; Cycle: *)
		tSA_Ign_2 : _tSAFICurrPmmREAL; (* Para: SAFI ignition current / duration setting 2 *) (* OldName:SAFICurr2PMM; Cycle: *)
		tSA_Ign_3 : _tSAFICurrPmmREAL; (* Para: SAFI ignition current / duration setting 3 *) (* OldName:SAFICurr3PMM; Cycle: *)
		tSA_Ign_4 : _tSAFICurrPmmREAL; (* Para: SAFI ignition current / duration setting 4 *) (* OldName:SAFICurr4PMM; Cycle: *)
		tSA_Ign_5 : _tSAFICurrPmmREAL; (* Para: SAFI ignition current / duration setting 5 *) (* OldName:SAFICurr5PMM; Cycle: *)
		tSA_Ign_6 : _tSAFICurrPmmREAL; (* Para: SAFI ignition current / duration setting 6 *) (* OldName:SAFICurr6PMM; Cycle: *)
		rSA_PBC_Sensitivity : REAL; (*PARA [12144]: PBC sensor sensitivity [mV/bar] *) (* OldName:ssDMR_empf; Cycle: *)
		rSA_ResetPos : REAL; (*PARA [12148]: SAFI reset position *) (* OldName:ssPosResSA; Cycle: *)
		rSA_EarlTiIonization : REAL; (*PARA [12135]: earliest timing for ionization *) (* OldName:ucAdvTiIonPMM; Cycle: *)
		rSA_CoilType : REAL; (*PARA [12130]: coil type *) (* OldName:ucCoilType; Cycle: *)
		rSA_DelFailR : REAL; (*PARA [12131]: trip limit spark delay failure rate *) (* OldName:ucDelFailRPMM; Cycle: *)
		rSA_DeMagLvl : REAL; (*PARA [12132]: magnatism level decrease *) (* OldName:ucDeMagLvlPMM; Cycle: *)
		rSA_DurFailR : REAL; (*PARA [12133]: spark duration deviation failure rate *) (* OldName:ucDurFailR; Cycle: *)
		rSA_DurTol : REAL; (*PARA [12134]: spark duration deviation limit *) (* OldName:ucDurTol; Cycle: *)
		rSA_InMagLvl : REAL; (*PARA [12140]: magnatism level increase *) (* OldName:ucInMagLvlPmm; Cycle: *)
		rSA_MxSpPow : REAL; (*PARA [12143]: limit for spark power *) (* OldName:ucMxSpPowPMM; Cycle: *)
		iSA_PIValveType : INT; (*PARA [12147]: valve type (1=Woodward, 2= Hoerbiger)*) (* OldName:ucPIValveType; Cycle: *)
		rSA_RetTiIon : REAL; (*PARA [12149]: latest timing for ionization *) (* OldName:ucRetTiIonPMM; Cycle: *)
		rSA_SparkCurChar : REAL; (*PARA [12150]: spark current characteristic *) (* OldName:ucSparkCurChar; Cycle: *)
		rSA_SparkCurLev : REAL; (*PARA [12151]: spark current level *) (* OldName:ucSparkCurLev; Cycle: *)
		rSA_SpPOffTi : REAL; (*PARA [12153]: turn on/off ration for spark power *) (* OldName:ucSpPOffTiPMM; Cycle: *)
		rSA_SparkDuration : REAL; (*PARA [12152]: SAFI spark duration  *) (* OldName:usDurationPMM; Cycle: *)
		rSA_Eps : REAL; (*PARA [12136]: eps *) (* OldName:usEps; Cycle: *)
		rSA_IgnPwrLi : REAL; (*PARA [12138]: SAFI ignition  power limitation  *) (* OldName:usIgnPwrLi; Cycle: *)
		rSA_IgnPwrOut : REAL; (*PARA [12139]: power supply output *) (* OldName:usIgnPwrOut; Cycle: *)
		rSA_MxIonMag : REAL; (*PARA [12141]: magnatism ionisation level *) (* OldName:usMxIonMagPMM; Cycle: *)
		rSA_MxMagLvl : REAL; (*PARA [12142]: magnatism level limit *) (* OldName:usMxMagLvlPMM; Cycle: *)
		rSA_IgnFeedbackLim : REAL; (*PARA [12137]: Time for ignition feedback *) (* OldName:usZuVLimPMM; Cycle: *)
		rCA_Win1_B : REAL; (*PARA [12122]: beginn of window 1 in 1/10 deg.  *) (* OldName:WMF1_B; Cycle: *)
		rCA_Win1_D : REAL; (*PARA [12123]: duration of window 1 in 1/10 deg.  *) (* OldName:WMF1_D; Cycle: *)
		rCA_Win2_B : REAL; (*PARA [12124]: beginn of window 2 in 1/10 deg.  *) (* OldName:WMF2_B; Cycle: *)
		rCA_Win2_D : REAL; (*PARA [12125]: duration of window 2 in 1/10 deg.  *) (* OldName:WMF2_D; Cycle: *)
		rCA_Win3_B : REAL; (*PARA [12126]: beginn of window 3 in 1/10 deg.  *) (* OldName:WMF3_B; Cycle: *)
		rCA_Win3_D : REAL; (*PARA [12127]: duration of window 3 in 1/10 deg.  *) (* OldName:WMF3_D; Cycle: *)
		rCA_Win4_B : REAL; (*PARA [14310]: beginn of window 4 in 1/10 deg.  *) (* OldName:WMF4_B; Cycle: *)
		rCA_Win4_D : REAL; (*PARA [14311]: duration of window 4 in 1/10 deg.  *) (* OldName:WMF4_D; Cycle: *)
		rSA_Win1_F : REAL; (*PARA [12154]: window 1 function *) (* OldName:FenstF1; Cycle: *)
		rSA_Win2_F : REAL; (*PARA [14312]: window 2 function *) (* OldName:FenstF2; Cycle: *)
		rSA_Win3_F : REAL; (*PARA [14313]: window 3 function *) (* OldName:FenstF3; Cycle: *)
		rSA_Win4_F : REAL; (*PARA [14314]: window 4 function *) (* OldName:FenstF4; Cycle: *)
		rU_IgnMon_LimActive : REAL; (*PARA [12155]: ignition voltage start monitoring  *) (* OldName:LimitActiv; Cycle: *)
		tIgn_LimitMonitor : ARRAY[0..4]OF _tMonicLimitREAL; (* Para: parameter voltage limit monitoring  *) (* OldName:LimitMon; Cycle: *)
		bIgn_LimitMonitorActive : ARRAY[0..4]OF BOOL; (* Para: type of voltage limit monitoring *) (* OldName:MonLimitOn; Cycle: *)
		bGridCode_Active : BOOL; (*PARA [11055]: Gride Code active *) (* OldName:bGridCode; Cycle: *)
		iEng_Motortype : INT; (* Para: Engine type *) (* OldName:motortyp; Cycle: *)
		bGridCodeMonitoringOnly : BOOL; (*PARA [11056]: Grid Code monitoring only active *) (* OldName:bGridCodeMonitoringOnly; Cycle: *)
		zz_V4_0_ParaVersionEnd : REAL := 4.0; (*! ADD NEW PARAMETER ONLY BELOW THIS LINE ! This is the end of base version parameter and has to stay unchanged. DO NOT CHANGE SORT ORDER of Para!*) (* OldName: new PV; Cycle: 5; *)
		rHCR : ARRAY[0..4]OF REAL; (* Para: Heat Capacity Ratio *) (* OldName: rKappa; Cycle: 2 *)
		bGT_SpecGasActive : BOOL; (*PARA [11374]: Sondergas *)
		bDynSparkDuration : BOOL; (*PARA [13646]: Variable spark duration active *) (* OldName:newPV; Cycle: *)
		usDurationIdle : UINT; (*PARA [13647]: Spark duration below power threshold *) (* OldName:newPV; Cycle: *)
		rP_Act_DynSpark_Limit_Nom : REAL; (*PARA [13648]: Spark duration below power threshold *) (* OldName:newPV; Cycle: *)
		iSA_CyclPIOnDuringMisf : USINT; (*PARA [13698]: Allowed Nr of cycles of ign off with PI on during misfire*) (* OldName:newPV; Cycle: *)
		rSA_PI_pudet_level : REAL; (*PARA [13699]: PI pull in current level *) (* OldName:newPV; Cycle: *)
		rSA_PI_pudet_st_time : REAL; (*PARA [13700]: PI pull in current start time *) (* OldName:newPV; Cycle: *)
		rSA_PI_pudet_duration : REAL; (*PARA [13701]: PI pull in current duration *) (* OldName:newPV; Cycle: *)
		rSA_PI_demag_delay : REAL; (*PARA [13707]: PI demagnetisation delay *) (* OldName:newPV; Cycle: *)
		rSA_PI_demag_duration : REAL; (*PARA [13708]: PI demagnetisation duration  *) (* OldName:newPV; Cycle: *)
		rSA_PI_demag_up_limit : REAL; (*PARA [13709]: PI demagnetisation upper limit *) (* OldName:newPV; Cycle: *)
		rSA_PI_currCtr_delay : REAL; (*PARA [13702]: PI correct current control delay *) (* OldName:newPV; Cycle: *)
		rSA_PI_currCtr_duration : REAL; (*PARA [13703]: PI correct current control duration *) (* OldName:newPV; Cycle: *)
		rSA_PI_currCtr_level : REAL; (*PARA [13704]: PI correct current control level *) (* OldName:newPV; Cycle: *)
		rSA_PI_currCtr_rate : REAL; (*PARA [13705]: PI correct current control failure rate *) (* OldName:newPV; Cycle: *)
		bPIDemagActive : BOOL; (*PARA [13706]: demagnetisation active *) (* OldName:newPV; Cycle: *)
		rSA_PI_clodet_st_time : ARRAY[0..24]OF REAL; (* PI close detection timing point *) (* OldName:newPV; Cycle: *)
		rSA_PI_clodet_set_current : REAL; (* PI close detection set point current *) (* OldName:newPV; Cycle: *)
		rSA_PI_clodet_set_duration : REAL; (* PI close detection set point duration *) (* OldName:newPV; Cycle: *)
		rSA_PI_clodet_duration : REAL; (* PI close detection duration *) (* OldName:newPV; Cycle: *)
		rSA_PI_clodet_cur_gradient : REAL; (* PI close detection current gradient *) (* OldName:newPV; Cycle: *)
		rSA_PI_clodet_var_limit_Start : REAL; (* PI close detection current gradient variation limit *) (* OldName:newPV; Cycle: *)
		rSA_PI_clodet_var_limit_Idle : REAL; (* PI close detection current gradient variation limit *) (* OldName:newPV; Cycle: *)
		rSA_PI_clodet_var_limit_Load : REAL; (* PI close detection current gradient variation limit *) (* OldName:newPV; Cycle: *)
		rSA_PI_curr1_current : REAL; (* PI set point 1 current *) (* OldName:newPV; Cycle: *)
		rSA_PI_curr1_duration : REAL; (* PI set point 1 duration *) (* OldName:newPV; Cycle: *)
		rSA_PI_curr2_current : REAL; (* PI set point 2 current *) (* OldName:newPV; Cycle: *)
		rSA_PI_curr2_duration : REAL; (* PI set point 2 duration *) (* OldName:newPV; Cycle: *)
		rSA_PI_curr3_current : REAL; (* PI set point 3 current *) (* OldName:newPV; Cycle: *)
		rSA_PI_curr3_duration : REAL; (* PI set point 3 duration *) (* OldName:newPV; Cycle: *)
		rSA_PI_curr4_current : REAL; (* PI set point 4 current *) (* OldName:newPV; Cycle: *)
		rSA_PI_recov_delay : REAL; (* PI energy recovery delay *) (* OldName:newPV; Cycle: *)
		rSA_PI_recov_current : REAL; (* PI energy recovery current *) (* OldName:newPV; Cycle: *)
		rSA_PI_recov_duration : REAL; (* PI energy recovery duration *) (* OldName:newPV; Cycle: *)
		iSA_NrOfMPM : USINT; (*PARA [14108]: SAFI number of  *) (* OldName:newPV; Cycle: *)
		bMORISonExh : BOOL; (*PARA [14352]: TRUE = MORIS rails are onto the exhaus pipes*)
		iU_EVCNoiseLim : UINT; (*PARA [14316]: Outlet valve closure noise limit*)
		iU_IVCNoiseLim : UINT; (*PARA [14317]: Inlet valve closure noise limit*)
		rNum_EVCThreshPer : REAL; (*PARA [14306]: Parameter for outlet valve closure detection*)
		rNum_IVCThreshPer : REAL; (*PARA [14307]: Parameter for inlet valve closure detection*)
		iU_EVCThreshMin : UINT; (*PARA [14308]: Minimum level for outlet valve closure detection*)
		iU_IVCThreshMin : UINT; (*PARA [14309]: Minimum level for inlet valve closure detection*)
		iKlS_MSFailure_Limit : UINT; (*PARA [12074]: limit for measuring signal failue [mV]*)
		bSA_Unb_Active : BOOL; (*PARA [14457]: Valve unbalance detection*)
		iCA_EVCDistLim : UINT; (*PARA [14458]: Maximum distance between the exhaust valve closure events*)
		iCA_IVCDistLim : UINT; (*PARA [14459]: Maximum distance between the intake valve closure events*)
		iCA_EarlyEVCLim : UINT; (*PARA [14460]: Valve unbalance detection exhaust valve closure timing minimum*)
		iCA_EarlyIVCLim : UINT; (*PARA [14461]: Valve unbalance detection intake valve closure timing minimum*)
		bKLS21_IgnMon : BOOL; (*PARA [14622]: KLS21 ignition monitoring*)
		iSA_PI_clodet_FailRLim : USINT; (*PARA [14623]: PI close detection failure rate limit [1/10 cycles]*)
		rNum_SAFI1_RelFwVer : REAL; (*PARA [14624]: Released SAFI1 firmware version*)
		rNum_SAFI2KLS_RelFwVer : REAL; (*PARA [14625]: Released SAFI2 KLS firmware version*)
		rNum_SAFI2DMR_RelFwVer : REAL; (*PARA [14626]: Released SAFI2 DMR firmware version*)
		rNum_SAFI3_RelFwVer : REAL; (*PARA [14627]: Released SAFI3 firmware version*)
		rNum_KLS21_RelFwVer : REAL; (*PARA [14628]: Released KLS21 firmware version*)
		rCA_KLS21_ITPDevLim : REAL; (*PARA [14629]: IP deviation limit [degCA]*)
		iNum_KLS21_ITPDevHist : USINT; (*PARA [14630]: Length of ignition events history [1/10 cycles]*)
		iNum_KLS21_ITPDevMax : USINT; (*PARA [14631]: Maximum missing ignition events [cycles]*)
		iNum_KLS21_ITPDevFailRLim : USINT; (*PARA [14632]: Failure rate limit for IP deviation [cycles]*)
		b_IgnIC_900Active : BOOL; (*PARA [12062]: TRUE=CAN ignition system is used *) (*OldName:ic900_vis; Cycle:;*)
		bSEMIC_Active : BOOL; (*PARA [14519]: Ignition controller SEMIC*)
		r_IgnIC_ResPosIC : REAL; (*PARA [12055]: Ignition reset pickup position *)
		rNum_PolEx : REAL; (*PARA [14900]: Polytropic exponent*)
		bFastStart_Act : BOOL; (* PARA [14184]: Fast Start package activated *)
	END_STRUCT;
END_TYPE
```

### module_SA.var - Package variables
```iecst
(********************************************************************
 * COPYRIGHT --
 ********************************************************************
 * File: Global.var
 * Author: BuR
 * Created: January 24, 2012
 ********************************************************************
 * Global variables of project Update
 ********************************************************************)
VAR
	bBlockCanUpdate : BOOL;
	AdvTimLi : INT; (* advanced ingnition timing 1/10 deg *)
	AussSchwel : UINT; (*not used OCA*)
	bACamSign : BOOL;
	bAMORISErr : BOOL;
	bAOverspeedErr : BOOL;
	bAParameter : BOOL;
	bAPICloseErr : BOOL;
	bAPIHardwareErr : BOOL;
	bAPIOpenErr : BOOL;
	bASAFIComErr : BOOL;
	bASAFIHwErr : BOOL;
	bASAFIWrongVers : BOOL;
	bATriggerSign : BOOL;
	bBCamSign : BOOL;
	bBCanErrRate : BOOL;
	bBConfigErr : BOOL;
	bBElectrTemp : BOOL;
	bBIgnPwrLim : BOOL;
	bBIGNShutOff : BOOL;
	bBIgnVoltMax : BOOL;
	bBIgnVoltMin : BOOL;
	bBMORISErr : BOOL;
	bBOffsetErr : BOOL;
	bBOutputErr : BOOL;
	bBOverspeedErr : BOOL;
	bBParameter : BOOL;
	bBPICloseErr : BOOL;
	bBPIHardwareErr : BOOL;
	bBPIOpenErr : BOOL;
	bBPIShutOff : BOOL;
	bBSAFIComErr : BOOL;
	bBSAFIFwErr : BOOL;
	bBSAFIHwErr : BOOL;
	bBSAFIWrongVers : BOOL;
	bBTriggerSign : BOOL;
	bGnlTrip1 : BOOL;
	bGnlTrip1_modlSA : BOOL;
	bGnlTrip2_modlSA : BOOL;
	bGnlTrip3_modlSA : BOOL;
	bGnlWarning_modlSA : BOOL;
	bWIgnPowerOverload : BOOL;
	bBIgnPowerOverload : BOOL;
	ucIgnPowerOverload : USINT;
	bAIgnPowerFail : BOOL;
	ucIgnPowerFail : USINT;
	bParaAct : BOOL;
	bPI_On : BOOL;
	bPIOpen : BOOL; (*response PI valve open*)
	bSAFI : ARRAY[0..12] OF _SAFIError;
	bSAFICfgMode : BOOL;
	bSAFIComErr : ARRAY[0..24] OF BOOL;
	bSAFIComm : BOOL;
	bSAFIConfig : BOOL;
	bSAFIError : ARRAY[0..12] OF _SAFIError; (* SAFI Error messages - CMS*)
	bSAFIIgnDisabRun : BOOL;
	bSAFIIgnDisabRunStat : BOOL;
	bSAFIIgnEnab : BOOL;
	bSAFIIgnEnabRun : BOOL;
	bSAFIPIDisabRun : BOOL;
	bSAFIPIDisabRunStat : BOOL;
	bSAFIPIEnab : BOOL;
	bSAFIPIEnabRun : BOOL;
	bSAFIReadStatus : BOOL;
	bSAFIRePara : ARRAY[0..12] OF BOOL;
	bSAFIReset : BOOL;
	bSAFISafetyLoop : BOOL;
	bSAFIStartComm : BOOL;
	bWCamSign : BOOL;
	bWCanErrRate : BOOL;
	bWConfigErr : BOOL;
	bWElectrTemp : BOOL;
	bWIgnPwrLim : BOOL;
	bWIgnVoltAvg : BOOL;
	bWIgnVoltDev : BOOL;
	bWIgnVoltMax : BOOL;
	bWIgnVoltMin : BOOL;
	bWOffsetErr : BOOL;
	bWOutputErr : BOOL;
	bWPIHardwareErr : BOOL;
	bWSAFIComErr : BOOL;
	bWSAFIFwErr : BOOL;
	bWTriggerSign : BOOL;
	CMSmain_SAFI_DMR : CMSmain;
	CMSmain_SAFI_Gen : CMSmain;
	CMSmain_SAFI_Ign : CMSmain;
	CMSmain_SAFI_KLS : CMSmain;
	CMSmain_SAFI_PI : CMSmain;
	CMSmain_SAFI_Gen_2 : CMSmain;
	CMSmain_SAFI_Ign_2 : CMSmain;
	CMSmain_SAFI_KLS_2 : CMSmain;
	CMSmain_SAFI_DMR_2 : CMSmain;
	CMSmain_SAFI_PI_2 : CMSmain;
	E_SAFI : ARRAY[0..12] OF _tEventSAFI; (* SAFI CAN Events *)
	EngType_SA : EngType;
	FenstF1 : USINT; (*Filter of KLS window 1*)
	FenstF2 : USINT; (*Filter of KLS window 2*)
	FenstF3 : USINT; (*Filter of KLS window 3*)
	FenstF4 : USINT; (*Filter of KLS window 4*)
	FenstF5 : USINT; (*Filter of KLS window 5*)
	FenstF6 : USINT; (*Filter of KLS window 6*)
	FireOrder : ARRAY[0..24] OF USINT;
	IN_SA : IN_SA_struct;
	KLS_md00 : ARRAY[0..12] OF _tSAFImdatas; (* KLS mdatas 0 *)
	KLS_md01 : ARRAY[0..12] OF _tSAFImdatas; (* KLS mdatas 1 *)
	KLS_md02 : ARRAY[0..12] OF _tSAFImdatas; (* KLS mdatas 2 *)
	KLS_md03 : ARRAY[0..12] OF _tSAFImdatas; (* KLS mdatas 3 *)
	KLS_md04 : ARRAY[0..12] OF _tSAFImdatas; (* KLS mdatas 4 *)
	KLS_md05 : ARRAY[0..12] OF _tSAFImdatas; (* KLS mdatas 5 *)
	KLS_md06 : ARRAY[0..12] OF _tSAFImdatas; (* KLS mdatas 6*)
	KLS_md07 : ARRAY[0..12] OF _tSAFImdatas; (* KLS mdatas 7*)
	KLSGW1 : UINT;
	KLSGW2 : UINT;
	KLSGW3 : UINT;
	KLSGW4 : UINT;
	LimitActiv : REAL;
	LimitMon : ARRAY[0..4] OF _tMonicLimit;
	MissfCyl : UDINT; (*cylinder misfire parameter*)
	MM2VIS : tMM2VIS;
	OpMode_SA : OpMode;
	OUT_SA : OUT_SA_struct;
	OvrSpeed : UINT; (* ignition overspeed parameter *)
	ParaFactoryDefault : Para_SA_struct; (*Test Init*)
	Para : Para_SA_struct;
	pm : Para_SA_struct;
	RetTimLi : INT; (* ignition retard timing limit *)
	SAFI : ARRAY[0..12] OF tSAFI;
	SAFI_md00 : ARRAY[0..12] OF _tSAFImdatas; (* SAFI mdatas 0 *)
	SAFI_md01 : ARRAY[0..12] OF _tSAFImdatas; (* SAFI mdatas 1 *)
	SAFI_md02 : ARRAY[0..12] OF _tSAFImdatas; (* SAFI mdatas 2 *)
	SAFI_md03 : ARRAY[0..12] OF _tSAFImdatas; (* SAFI mdatas 3 *)
	SAFI_md04 : ARRAY[0..12] OF _tSAFImdatas; (* SAFI mdatas 4 *)
	SAFI_md05 : ARRAY[0..12] OF _tSAFImdatas; (* SAFI mdatas 5 *)
	SAFICurr0 : _tSAFICurr; (* SAFI current/duration setting 7 *)
	SAFICurr0PMM : _tSAFICurrPmm;
	SAFICurr0Sel : _tSAFICurrPmm;
	SAFICurr1 : _tSAFICurr; (* SAFI current/duration setting 1 *)
	SAFICurr1PMM : _tSAFICurrPmm; (* SAFI current/duration setting 2 *)
	SAFICurr2 : _tSAFICurr; (* SAFI current/duration setting 2 *)
	SAFICurr2PMM : _tSAFICurrPmm; (* SAFI current/duration setting 2 *)
	SAFICurr3 : _tSAFICurr; (* SAFI current/duration setting 3 *)
	SAFICurr3PMM : _tSAFICurrPmm; (* SAFI current/duration setting 3 *)
	SAFICurr4 : _tSAFICurr; (* SAFI current/duration setting 4 *)
	SAFICurr4PMM : _tSAFICurrPmm; (* SAFI current/duration setting 5 *)
	SAFICurr5 : _tSAFICurr; (* SAFI current/duration setting 5 *)
	SAFICurr5PMM : _tSAFICurrPmm; (* SAFI current/duration setting 5 *)
	SAFICurr6 : _tSAFICurr; (* SAFI current/duration setting 6 *)
	SAFICurr6PMM : _tSAFICurrPmm; (* SAFI current/duration setting 6 *)
	SAFIError : ARRAY[0..12] OF _SAFIError; (* SAFI Error messages *)
	slTiming : ARRAY[0..12] OF DINT;
	ssDMR_empf : INT; (*Empfindlichkeit DMR Sensoren [mV/bar]*)
	ssNEf : INT; (* DMR Niveaueinpassung fein *)
	ssNEg : INT; (* DMR Niveaueinpassung grob *)
	ssPosResSA : INT; (* SAFI reset position *)
	ssSAFITemp : ARRAY[0..12] OF INT;
	ssSAFMaxT : ARRAY[0..12] OF INT;
	ssWEf : INT; (* DMR Winkeleinpassung fein *)
	ssWEg : INT; (* DMR Winkeleinpassung grob *)
	ucAdvTiIon : USINT;
	ucAdvTiIonPMM : USINT;
	ucAussInt : USINT; (* DMR Intervall Aussetzer *)
	ucCamSign : USINT;
	ucCanErrRate : USINT;
	ucCoilType : USINT; (*Coil type*)
	ucConfigErr : USINT;
	ucConfigState : USINT;
	ucDelFailR : USINT;
	ucDelFailRPMM : USINT;
	ucDeMagLvl : USINT;
	ucDeMagLvlPMM : USINT;
	ucDurFailR : USINT;
	ucDurTol : USINT;
	ucElectrTemp : USINT;
	ucEmpf : ARRAY[0..13] OF USINT;
	ucERDurTol : ARRAY[0..24] OF USINT; (* Error Rate for Duration Tolerance *)
	ucERZuV : ARRAY[0..24] OF USINT; (* Error Rate for spark delay *)
	ucFuAU : USINT; (* DMR Funk. Aussetzer *)
	ucFuGZ : USINT; (* DMR Funk. Gluezuenden *)
	ucFuIM : USINT; (* DMR Funk. Indiz. Mitteldruck *)
	ucFuNAE : USINT; (* DMR Funk. NOx Aequivalent *)
	ucFuNE : USINT; (* DMR Funk. Niveaueinpassung *)
	ucFuVL : USINT; (* DMR Funk. Verbrennungslage *)
	ucFuWE : USINT; (* DMR Funk. Winkeleinpassung *)
	ucIGNMode : ARRAY[0..12] OF USINT; (* SAFI-IGN Mode *)
	ucIgnPwrLim : USINT;
	ucIGNShutOff : USINT;
	ucIgnVoltMax : USINT;
	ucIgnVoltMin : USINT;
	ucInMagLvl : USINT;
	ucInMagLvlPMM : USINT;
	ucIonis : USINT;
	ucKLSMode : ARRAY[0..12] OF USINT;
	ucKuA : USINT; (* DMR Kurvenart *)
	ucMORISErr : USINT;
	ucMxSpPow : USINT;
	ucMxSpPowPMM : USINT;
	ucNrOfFiringCyl : USINT;
	ucNumberOfCylinder : USINT;
	ucOffsetErr : USINT;
	ucOutputErr : USINT;
	ucOverspeedErr : USINT;
	ucParameter : USINT;
	ucPICloseErr : USINT;
	ucPIHardwareErr : USINT;
	ucPIOpenErr : USINT;
	ucPIShutOff : USINT;
	ucReParaState : ARRAY[0..12] OF USINT;
	ucRetTiIon : USINT;
	ucRetTiIonPMM : USINT;
	ucSAFIComErr : USINT;
	ucSAFIConf : ARRAY[0..12] OF USINT; (* SAFI I/O rotation *)
	ucSAFIFwErr : USINT;
	ucSAFIHwErr : USINT;
	ucSAFIMode : ARRAY[0..12] OF USINT;
	ucSAFIWrongVers : USINT;
	ucSparkCurChar : USINT; (*Sparkc characteristic*)
	ucSparkCurLev : USINT; (*Spark current level*)
	ucSpPOffTi : USINT;
	ucSpPOffTiPMM : USINT;
	ucTriggerSign : USINT;
	ucUP_Pos : USINT;
	ulProdDate : ARRAY[0..12] OF _tSAFIProdDate;
	ulSAFArbH : ARRAY[0..12] OF UDINT;
	ulSAFBetrH : ARRAY[0..12] OF UDINT; (* SAFI Betriebsstunden *)
	ulSAFSerNr : ARRAY[0..12] OF UDINT;
	ulZuendEin : UDINT; (* actual cylinder firing state *)
	usAbstAB : UINT;
	usAbstBA : UINT;
	usAussGW : UINT; (* DMR GW Aussetzer *)
	usAussTmax : UINT := 2000;
	usBohr : UINT;
	usDMRMode : ARRAY[0..12] OF UINT;
	usDuration : ARRAY[0..1] OF UINT; (* SAFI spark duration *)
	usDurationPMM : UINT; (* SAFI spark duration *)
	usEps : UINT;
	usErrZahnz : ARRAY[0..12] OF UINT;
	usErrZykl : UINT;
	usGluehGW : UINT; (* DMR GW Gluehzuenden *)
	usHub : UINT;
	usIgnPwrLi : UINT; (* SAFI Ignition Power limitation *)
	usIgnPwrOut : UINT; (*power supply output*)
	usIgnPwrPMM : UINT;
	usIPEx : UINT; (* DMR Iterativer Polytropenexponent *)
	usIPFa : UINT; (* DMR It. Polytropenexpo Faktor *)
	usIPGr : UINT; (* DMR It. Polytropenexpo Grenzwert *)
	usIPIt : UINT; (* DMR It. Polytropenexpo It. grenze *)
	usIPKo : UINT; (* DMR It. Polytropenexpo Korrektur *)
	usKlopfGW : UINT; (* DMR GW Klopfen *)
	usMode : ARRAY[0..12] OF UINT;
	usMW_KLS1 : UINT; (*Average #kls__mdatas1 MUX 0/1 [cycles]*)
	usMW_KLS2 : UINT; (*Average #kls__mdatas1 MUX 2/3 [cycles]*)
	usMW_KLS3 : UINT; (*Average #kls__mdatas1 MUX 4/5 [cycles]*)
	usMW_KLS4 : UINT; (*Average #kls__mdatas1 MUX 6/7 [cycles]*)
	usMWEr : UINT; (* DMR Mittelwert Erweitert *)
	usMWNGA : UINT; (* DMR MW Niveaueinp, Gluehz, Aussetz *)
	usMWSt : UINT; (* DMR MW Statistik *)
	usMxIonMag : UINT;
	usMxIonMagPMM : UINT;
	usMxMagLvl : UINT;
	usMxMagLvlPMM : UINT;
	usNennDz : UINT; (* DMR Nenndrehzahl *)
	usNETol : UINT; (* DMR Niveaueinpassung Toleranz *)
	usPleuel : UINT;
	usPolEx : UINT; (* DMR Iterativer Polytropenexponent *)
	usSAFFiltV : ARRAY[0..12] OF UINT; (*SAFI KLS filter version*)
	usSAFIHW : ARRAY[0..12] OF _tSAFIHardware; (* SAFI Hardwareversion *)
	usSAFIVers : ARRAY[0..12] OF UINT; (* SAFI Firmwareversion *)
	usSAFIVersMin : UINT;
	usStartHP : UINT;
	usthVW : UINT; (* DMR thermodyn. Verlustwinkel *)
	usTolZZP : UINT;
	usVLFa : UINT; (* DMR Verbrennungslage Faktor *)
	usWMA_B : UINT; (* DMR Winkelfensterbeginn Aussetzer *)
	usWMA_D : UINT; (* DMR Winkelfensterdauer Aussetzer *)
	usWMBB_B : UINT; (* DMR WFbeginn Brennbeginn *)
	usWMBB_D : UINT; (* DMR WFdauer Brennbeginn *)
	usWMBD_B : UINT; (* DMR WFbeginn Brenndauer *)
	usWMBD_D : UINT; (* DMR WFdauer Brenndauer *)
	usWMG_B : UINT; (* DMR Winkelfensterbeginn Gluehzuend *)
	usWMG_D : UINT; (* DMR Winkelfensterdauer Gluezuenden *)
	usWMK_B : UINT; (* DMR Winkelfensterbeginn Klopfen *)
	usWMK_D : UINT; (* DMR Winkelfensterdauer Klopfen *)
	usWMNEf_B : UINT; (* DMR WFbeginn Niveaueinp. fein *)
	usWMNEf_D : UINT; (* DMR WFdauer Niveaueinp. fein *)
	usWMNEg_B : UINT; (* DMR WFbeginn Niveaueinp. grob *)
	usWMNEg_D : UINT; (* DMR WFdauer Niveaueinp. grob *)
	usWMS_B : UINT; (* DMR Winkelfensterbeginn Sp. druck *)
	usWMS_D : UINT; (* DMR Winkelfensterdauer Sp. druck *)
	usWMVL1_B : UINT; (* DMR WFbeginn Verbrennungslage Art1 *)
	usWMVL1_D : UINT; (* DMR WFdauer Verbrennungslage Art1 *)
	usWMWE_B : UINT; (* DMR WFdauer Winkeleinpassung *)
	usWMWE_D : UINT; (* DMR WFbeginn Winkeleinpassung *)
	usZahnzahl : UINT;
	usZuVLim : UINT;
	usZuVLimPMM : UINT;
	VIS2MM : tVIS2MM;
	WMF_AB : UINT; (*not used OCA*)
	WMF_AD : UINT := 50; (*not used OCA*)
	WMF1_B : UINT; (* Start of window 1 [degCA]*)
	WMF1_D : UINT; (* Duration of window 1 [degCA] *)
	WMF2_B : UINT; (* Start of window 2 [degCA]*)
	WMF2_D : UINT; (* Duration of window 2 [degCA]*)
	WMF3_B : UINT; (* Start of window 3 [degCA]*)
	WMF3_D : UINT; (* Duration of window 3 [degCA]*)
	WMF4_B : UINT; (* Start of window 4 [degCA]*)
	WMF4_D : UINT := 50; (* Duration of window 4 [degCA]*)
	WMF5_B : UINT; (* Start of window 5 [degCA]*)
	WMF5_D : UINT := 1; (* Duration of window 5 [degCA]*)
	WMF6_B : UINT; (* Start of window 6 [degCA]*)
	WMF6_D : UINT := 1; (* Duration of window 6 [degCA]*)
	ZylZahl : USINT;
	bAPBCMemBurst : BOOL;
	bBPBCMemBurst : BOOL;
	ucPBCMemBurst : USINT;
	bWPBCCompLineCheck : BOOL;
	bBPBCCompLineCheck : BOOL;
	ucPBCCompLineCheck : USINT;
	bWPBCNegVoltCheck : BOOL;
	bBPBCNegVoltCheck : BOOL;
	ucPBCNegVoltCheck : USINT;
	bWPBCNegPresCheck : BOOL;
	bBPBCNegPresCheck : BOOL;
	ucPBCNegPresCheck : USINT;
	bWPBCPresSlopeCheck : BOOL;
	bBPBCPresSlopeCheck : BOOL;
	ucPBCPresSlopeCheck : USINT;
	bWPBCSlowDriftCheck : BOOL;
	bBPBCSlowDriftCheck : BOOL;
	ucPBCSlowDriftCheck : USINT;
	bWPBCConfNotOK : BOOL;
	bBPBCConfNotOK : BOOL;
	ucPBCConfNotOK : USINT;
	bAPBCSensErr : BOOL;
	bBPBCSensErr : BOOL;
	ucPBCSensErr : USINT;
	bWPBCInvalidPar : BOOL := FALSE;
	bBPBCInvalidPar : BOOL := FALSE;
	ucPBCInvalidPar : USINT := 0;
	bWMORISErr : BOOL;
	ucCountG : USINT;
	bNoInitDetected : BOOL := FALSE; (*allways true, except 1cycle on init up*)
	SIM_rN_IgnSAFI_Act : REAL; (* Engine speed measured by ignition SAFI *)
	SIM_rT_EG_Cyl : ARRAY[0..24] OF REAL; (* cylinder exhaust gas temperatures *)
	SIM_iU_SAFI_Win1 : ARRAY[0..24] OF INT; (* cylinder values of KLS window 1 *)
	SIM_iU_SAFI_Win2 : ARRAY[0..24] OF INT; (* cylinder values of KLS window 2 *)
	SIM_rU_IgnSAFI_Max : REAL; (* maximum ignition voltage  *)
	SIM_rU_IgnSAFI_Min : REAL; (* minimum ignition voltage  *)
	SIM_rU_IgnSAFI_Cyl : ARRAY[0..24] OF REAL; (* ignition voltage for each cylinder  *)
	SIM_rU_IgnSAFI_Avg : REAL; (* ignition voltage average *) (* OldName:AvgVolt; Cycle:5 *)
	usIgnPwr : UINT;
	DMR_Ref : tDMR_ref;
	ucUpCur : ARRAY[0..12] OF USINT;
	ssWEf_L : ARRAY[0..25] OF INT;
	ssWEf_H : ARRAY[0..25] OF INT;
	DMR_cur : ARRAY[0..12] OF _tSAFImdatas;
	bAPBCCPSSat : BOOL; (*Cylinder pressure saturation trip*)
	bBPBCCPSSat : BOOL; (*Cylinder pressure saturation message*)
	ucPBCCPSSat : USINT; (*Cylinder pressure saturation cyl info*)
	ucNrCyPiMf : USINT; (*Allowed Nr of cycles of ign off with PI on during misfire*)
	bAPIDemagFail : BOOL;
	bBPIDemagFail : BOOL;
	ucPIDemagFail : USINT;
	bWPICurrCtrWarn : BOOL;
	bBPICurrCtrWarn : BOOL;
	ucPICurrCtrWarn : USINT;
	bAPICurrCtrRate : BOOL;
	Diag : ARRAY[0..12] OF tDiag;
	bParaActCyl : ARRAY[0..24] OF BOOL;
	CMSinit_SAFI_x_status : UINT; (* CAN SAFI Module Init Status *)
	CMSmain_SAFI_x_status : UINT; (* CAN SAFI Module Main Status *)
	ssPIvar_limt_Idle : INT;
	ssPIvar_limt_Load : INT;
	ssPIvar_limt_Start : INT;
	ssPICurGradStart : INT;
	bMORIS_OnEx : BOOL; (*True = MORIS on Exhaust*)
	bAExValveErr : BOOL;
	bBExValveErr : BOOL;
	iIdx_ExValveErr : USINT;
	bAInValveErr : BOOL;
	bBInValveErr : BOOL;
	iIdx_InValveErr : USINT;
	iMisfCylPICloDet : UDINT; (*cylinder misfire parameter from PI close detection*)
	PICurGrad : ARRAY[0..24] OF tPICurGrad;
	bWExValveUnb : BOOL;
	bBExValveUnb : BOOL;
	iIdx_ExValveUnb : USINT;
	bWInValveUnb : BOOL;
	bBInValveUnb : BOOL;
	iIdx_InValveUnb : USINT;
	bSA_Win1Frozen : ARRAY[0..24] OF BOOL; (*Knock noise signal  frozen*)
	bSA_Win1Altern : ARRAY[0..24] OF BOOL; (*Knock noise signal alternating*)
	bWSAFrozenAltern : BOOL;
	bBSAFrozenAltern : BOOL;
	iIdx_SAFrozenAltern : USINT;
	bSA_U_CylFrozen : ARRAY[0..24] OF BOOL; (*Ignition voltage frozen*)
	bSA_U_CylAltern : ARRAY[0..24] OF BOOL; (*Ignition voltage alternating*)
	bSA_PmaxFrozen : ARRAY[0..24] OF BOOL; (*DMR knock signal frozen*)
	bSA_PmaxAltern : ARRAY[0..24] OF BOOL; (*DMR knock signal alternating*)
	bSA_IMEP_Frozen : ARRAY[0..24] OF BOOL; (*IMEP frozen*)
	bSA_IMEP_Altern : ARRAY[0..24] OF BOOL; (*IMEP alternating*)
	bSA_PICurGradFrozen : ARRAY[0..24] OF BOOL; (*PI close current gradient frozen*)
	bSA_PICurGradAltern : ARRAY[0..24] OF BOOL; (*PI close current gradient alternating*)
	iNum_UpCurKls : USINT; (*Curve upload memory allocation - Percentage of KLS data [%]*)
	iCA_ITP_DevLim : USINT; (*ITP deviation limit [degCA * 10]*)
	iNum_ITP_DevFailR : USINT; (*Failure rate limit for ITP deviation [1 / 10 cycles]*)
	iNum_LenIgnHist : USINT; (*Length of ignition events history [cycles]*)
	iNum_IgnMiss_Max : USINT; (*Maximum missing ignition events [cycles]*)
	iNum_UpCurKlsSet : USINT; (*KLS up curve settings*)
	bW_KLS21_NoIgnMon : BOOL; (*W9350 - KLS21 ignition monitoring not available*)
	bB_KLS21_NoIgnMon : BOOL; (*B9050 - KLS21 ignition monitoring not available*)
	iIdx_KLS21_NoIgnMon : USINT; (*B9050 - KLS21 ignition monitoring not available - cylinder number*)
	bSAFIErrorReset : BOOL;
	bUnknownDevice : BOOL; (*At least one unknown device is installed*)
	bSAFI1 : BOOL; (*At least one SAFI1 is installed*)
	bSAFI2KLS : BOOL; (*At least one SAFI2KLS is installed*)
	bSAFI2DMR : BOOL; (*At least one SAFI2DMR is installed*)
	bSAFI3 : BOOL; (*At least one SAFI3 is installed*)
	bKLS21 : BOOL; (*At least one KLS21 is installed*)
	bSAFI3_all : BOOL; (*All devices are SAFI3*)
	rTi_MaxSkipFire : REAL; (*Maximum time for skipfire operation [s]*)
	iCA_StartHPWin : UINT; (*Start of high pressure window [degCA]*)
	ucRelCheckState : USINT;
END_VAR
```

### Program Logical/SAFI/safi_spd (IEC, version 4.07.0) - + SAFI speed measurement

- safi_spdCyclic.st (not readable text: treated as protected, skipped)

#### safi_spd.var
```iecst
(********************************************************************
 * COPYRIGHT -- INNIO Company
 ********************************************************************
 * Program: safi_spd
 * File: safi_spd.var
 * Author: 105026877
 * Created: July 14, 2015
 ********************************************************************
 * Local variables of program safi_spd
 ********************************************************************)
VAR
	SafiSpeedSumm : UDINT;
	ucCylIndex : USINT;
	ucSpeedAvgCount : USINT;
	usNoSpeedCount : UINT;
	SAFISpeed : ARRAY[0..24] OF _tSAFISpeed;
	LCCounter_0 : LCCounter;
	slTest1 : DINT;
	slTest2 : DINT;
	ssInternalFactor : INT;
	usHelpA : UINT := 100;
	TOF_NetpM : TOF;
	n_lastValOK : UINT;
END_VAR
```

### Program Logical/SAFI/safi_gen (IEC, version 4.14.0) - + SAFI general

- safi_genCyclic.st (not readable text: treated as protected, skipped)

- safi_genInit.st (not readable text: treated as protected, skipped)

#### safi_gen.var
```iecst
VAR
	AmmSeqCamSign : AmmSequence;
	AmmSeqCanErrRate : AmmSequence;
	AmmSeqConfigErr : AmmSequence;
	AmmSeqElectrTemp : AmmSequence;
	AmmSeqFwErr : AmmSequence;
	AmmSeqHwErr : AmmSequence;
	AmmSeqMORISErr : AmmSequence;
	AmmSeqParaErr : AmmSequence;
	AmmSeqSAFIComErr : AmmSequence;
	AmmSeqTriggerSign : AmmSequence;
	AmmSeqWrongVers : AmmSequence;
	bAmmSeqClkP : BOOL;
	bCamSign : ARRAY[0..24] OF BOOL;
	bCanErrRate : ARRAY[0..24] OF BOOL;
	bConfigErr : ARRAY[0..24] OF BOOL;
	bElectrTemp : ARRAY[0..24] OF BOOL;
	bFwError : ARRAY[0..24] OF BOOL;
	bHwError : ARRAY[0..24] OF BOOL;
	bIPDeviation : ARRAY[0..24] OF BOOL;
	bMORISErr : ARRAY[0..24] OF BOOL;
	bParaErr : ARRAY[0..24] OF BOOL;
	bToggle : BOOL;
	bToggle_Old : ARRAY[0..24] OF BOOL;
	bTriggerSign : ARRAY[0..24] OF BOOL;
	bVersionMonAct : BOOL;
	bWrongVers : ARRAY[0..24] OF BOOL;
	TOF_VersMon : TOF;
	TON_100msTick : TON;
	TON_SecondTick : TON;
	ucCylIndex : USINT;
	ucNodeCount : USINT;
	ucNrOfFaults : USINT;
	ucResetState : USINT;
	ucTimingCounter : USINT;
	usCamErrCnt : ARRAY[0..24] OF UINT;
	usErrZyklOld : UINT;
	usEventSum : UINT;
	usTolZZPOld : UINT;
	usTriggerErrCnt : ARRAY[0..24] OF UINT;
	bParaSendOK : BOOL;
	SAFI_tPI_tPIopenH_old : ARRAY[0..12] OF tPIopen;
	ucSAFIPIParaSend : USINT;
	SAFI_tPI_tPIopenL_old : ARRAY[0..12] OF tPIopen;
	usEventSum2 : UINT;
	bParaSendOK2 : BOOL;
	ucReDoCount2 : USINT;
	ucToggle : USINT;
	TON_50msTick : TON;
	TON_CANGo : TON;
	AmmSeqPBCMemBurst : AmmSequence;
	AmmSeqPBCCPSSat : AmmSequence := (0); (*Amm sequence for CPS saturation*)
	AmmSeqPBCCompLineCheck : AmmSequence;
	AmmSeqPBCNegVoltCheck : AmmSequence;
	AmmSeqPBCNegPresCheck : AmmSequence;
	AmmSeqPBCPresSlopeCheck : AmmSequence;
	AmmSeqPBCSlowDriftCheck : AmmSequence;
	AmmSeqPBCConfNotOK : AmmSequence;
	AmmSeqPBCInvalidPar : AmmSequence;
	AmmSeqPBCSensErr : AmmSequence;
	ssPBCMemBurst : ARRAY[0..24] OF INT;
	bTEST_BURST : ARRAY[0..24] OF BOOL;
	bTEST_CPSSat : ARRAY[0..24] OF BOOL := [25(0)]; (*Test flags for the CPS saturation*)
	bPBCSensErr : ARRAY[0..24] OF BOOL;
	TON_SensErr : ARRAY[0..24] OF TON;
	bPBCSensErrTest : ARRAY[0..24] OF BOOL;
	ssMotorzyklus : INT;
	ssPBCMemBurstLimit : INT;
	usCount : UINT;
	ucCylNum : USINT;
	usResetCnt : UINT;
	ssTimingOld : INT;
	bTrigger_ITPSend : BOOL;
	SAFI_tPI_Mode_old : ARRAY[0..24] OF UINT;
	iPICurGradDiff : ARRAY[0..24] OF INT;
	iCntPIclodet : ARRAY[0..24] OF INT;
	bTripPIclodet : BOOL;
	iPICurGradOld : ARRAY[0..24] OF INT;
	bCloseErr : ARRAY[0..24] OF BOOL;
	AmmSeqCloseErr : AmmSequence;
	TON_CloseErrReset : TON;
	TON_Load_Delay : TON;
	iCntPInoclodet : ARRAY[0..24] OF USINT;
	tPIclodet5_old : ARRAY[0..12] OF tPIclosdet5;
	rP_Red_SAComErr_Norm : REAL; (*Power redution if half or more SAFI have a CAN communication failure*)
	rP_Red_SARebootErr_Norm : REAL; (*Power reduction if a SAFI rebooted too often*)
	bTPIN_SAFIReboot : ARRAY[0..12,0..2] OF BOOL; (*Input of timer for max allowed of SAFI reboots rate*)
	iCnt_SAFIReboot : ARRAY[0..12] OF USINT; (*Counter for timer for max allowed SAFI reboot rate*)
	xTP_SAFIReboot : ARRAY[0..12,0..2] OF TP;
	xF_TRIG_SAFIReboot : ARRAY[0..12] OF F_TRIG;
	xTP_P_Red_SAFIReboot : TP;
	iCnt_IndexDim2 : USINT;
	iCnt_FaultsSAFIComErr : USINT;
	bSAFISendAllPara : BOOL;
	bSAFISendAllPIParaTC1 : BOOL;
	ssTiming : ARRAY[0..24] OF INT;
	ucSAFIModeOld : ARRAY[0..12] OF USINT;
	ucSAFIParaSend : USINT;
	bSA_FrozenAltern : ARRAY[0..24] OF BOOL;
	rT_EG_Cyl_old1 : ARRAY[0..24] OF REAL;
	rT_EG_Cyl_old2 : ARRAY[0..24] OF REAL;
	xTON_T_EG_CylFrozen : ARRAY[0..24] OF TON;
	xTON_T_EG_CylAltern : ARRAY[0..24] OF TON;
	bSA_T_EGCylFrozen : ARRAY[0..24] OF BOOL; (*Exhaust gas temperature forzen*)
	bSA_T_EGCylAltern : ARRAY[0..24] OF BOOL; (*Exhaust gas temperature alternating*)
	AmmSeqSAFIFrozenAltern : AmmSequence;
	xTON_SAFIFroAltReset : TON;
	bSA_FrozenAltern_All : BOOL;
	xTON_SACfgDone : TON; (*Timer to set A3333 if a SAFI is not in operation mode for too long*)
	iNum_UpCurKlsOld : USINT; (*Curve upload memory allocation - Percentage of KLS data [%] - Old*)
	bNoKLS21IgnMon : ARRAY[0..24] OF BOOL; (*Para KLS21 ignition monitoring is rue but device is not a KLS21*)
	AmmSeqNoKLS21IgnMon : AmmSequence;
	SAFI_tPI_tPIopenH_diff : ARRAY[0..12] OF INT;
	SAFI_tPI_tPIopenL_diff : ARRAY[0..12] OF INT;
END_VAR
```

### Program Logical/SAFI/safi_mod (IEC, version 4.14.0) - + SAFI mode

- safi_modCyclic.st (not readable text: treated as protected, skipped)

#### safi_mod.var
```iecst
VAR CONSTANT
	PowerUp : USINT := 0;
	Configuration : USINT := 10;
	Operation : USINT := 20;
	SelfTest : USINT := 30;
	Reset : USINT := 40;
END_VAR
VAR
	bDelayReset : BOOL;
	TON_Reset : TON;
	ucCylIndex : UINT;
	ucSAFIState : USINT;
END_VAR
```

### Program Logical/SAFI/safi_cfg (IEC, version 4.14.0) - + SAFI config

- safi_cfgCyclic.st (not readable text: treated as protected, skipped)

- safi_cfgInit.st (not readable text: treated as protected, skipped)

#### safi_cfg.var
```iecst
VAR
	ucSAFIConfCnt : USINT;
	usCheckXor : UINT;
	usCheckXorOld : UINT;
	ulCheckSum : UDINT;
	ulCheckSumOld : UDINT;
	TON_SecondTick : TON;
	ucCylIndex : USINT;
	ucStatusCnt : USINT;
	ucReParaCount : ARRAY[0..12] OF USINT;
	usEvery10SecOneSAFI : UINT;
	ucHelp : USINT;
	usWait : ARRAY[0..12] OF UINT;
	usReParaDuration : ARRAY[0..12] OF UINT;
	ucReParaCycl : ARRAY[0..12] OF USINT;
END_VAR
```

### Program Logical/SAFI/safi_hs (IEC, version 4.12.0) - + SAFI high voltage measurement

- safi_hsCyclic.st (not readable text: treated as protected, skipped)

#### safi_hs.var
```iecst
VAR
	TON_SecondTick : TON; (* CAN VUS FAHLER *)
	ucCylIndex : USINT;
	ucMonDiffCnt : USINT;
	ucMonMinCnt : ARRAY[0..24] OF USINT;
	ucMonMaxCnt : ARRAY[0..24] OF USINT;
	ucMonAvgCnt : USINT;
	AmmSeqIgnVoltMax : AmmSequence;
	AmmSeqIgnVoltMin : AmmSequence;
	bAmmSeqClkP : BOOL;
	bOffsetErr : ARRAY[0..24] OF BOOL;
	AmmSeqOffsetErr : AmmSequence;
	rAvgVoltSum : REAL;
	rU_Cyl : ARRAY[0..24] OF REAL;
	bIgnVoltMin : ARRAY[0..24] OF BOOL;
	bIgnVoltMax : ARRAY[0..24] OF BOOL;
	rU_Cyl_old1 : ARRAY[0..24] OF REAL;
	rU_Cyl_old2 : ARRAY[0..24] OF REAL;
	xTON_U_CylFrozen : ARRAY[0..24] OF TON;
	xTON_U_CylAltern : ARRAY[0..24] OF TON;
END_VAR
```

### Program Logical/SAFI/safi_ign (IEC, version 4.14.0) - + SAFI ignition

- safi_ignCyclic.st (not readable text: treated as protected, skipped)

#### safi_ign.var
```iecst
VAR
	AdvTimLi_Old : INT;
	AmmSeqOutputErr : AmmSequence;
	AmmSeqOverspeedErr : AmmSequence;
	bAmmSeqClkP : BOOL;
	bOutputErr : ARRAY[0..24] OF BOOL;
	bOverspeedErr : ARRAY[0..24] OF BOOL;
	bToggle : BOOL;
	bToggle2 : BOOL;
	OvrSpeed_Old : UINT;
	RetTimLi_Old : INT;
	SAFICurr1_Old : _tSAFICurrPmm;
	SAFICurr2_Old : _tSAFICurrPmm;
	SAFICurr3_Old : _tSAFICurrPmm;
	SAFICurr4_Old : _tSAFICurrPmm;
	SAFICurr5_Old : _tSAFICurrPmm;
	SAFICurr6_Old : _tSAFICurrPmm;
	SAFICurr0_Old : _tSAFICurrPmm;
	TON_SecondTick : TON;
	TON_Selftest : TON;
	TON_TestDelay : TON;
	ucAdvTiIon_Old : USINT;
	ucCylCount : USINT;
	ucCylIndex : USINT;
	ucDeMagLvl_Old : USINT;
	ucDurTol_Old : USINT;
	ucDelFailR_Old : USINT;
	ucIGNMode_Old : ARRAY[0..12] OF USINT;
	ucInMagLvl_Old : USINT;
	ucIonis_Old : USINT;
	ucMxSpPow_Old : UINT;
	ucOutputErrCnt : USINT;
	ucReDoCount : USINT;
	ucRetTiIon_Old : USINT;
	ucSAFICheck : USINT;
	ucSpPOffTi_Old : USINT;
	usAussTmax_Old : UINT;
	usCheckTime : UINT;
	usDuration_Old : UINT;
	usEventSum : UINT;
	usIgnPwrLi_Old : UINT;
	usMxIonMag_Old : UINT;
	usMxMagLvl_Old : UINT;
	usZuVLim_Old : UINT;
	usCurrData : ARRAY[0..10] OF UINT;
	DatObjInfo_SAFICurr : DatObjInfo;
	ucSparkCurCharOld : USINT;
	DatObjRead_SAFICurr : DatObjRead;
	SAFICurr1Sel : _tSAFICurrPmm;
	SAFICurr2Sel : _tSAFICurrPmm;
	SAFICurr3Sel : _tSAFICurrPmm;
	SAFICurr4Sel : _tSAFICurrPmm;
	SAFICurr5Sel : _tSAFICurrPmm;
	SAFICurr6Sel : _tSAFICurrPmm;
	DatObjRead_CoilType : DatObjRead;
	DatObjInfo_CoilType : DatObjInfo;
	ucCoilTypeOld : USINT;
	usCoilData : ARRAY[0..12] OF UINT;
	bParaSendOK : BOOL;
	bIgnPwrLim : ARRAY[0..24] OF BOOL;
	AmmSeqIgnPwrLim : AmmSequence;
	ucDurFailR_Old : USINT;
	bArnoMan : BOOL;
	bCheck : BOOL;
	bSAFISendAllIGNPara : BOOL;
	ssActTiming : ARRAY[0..24] OF INT; (* actual timing measured *)
	ucSAFIIgnParaSend : USINT;
	iCA_ITP_DevLim_Old : USINT; (*ITP deviation limit [degCA * 10] - Old*)
	iNum_ITP_DevFailR_Old : USINT; (*Failure rate limit for ITP deviation [1 / 10 cycles] - Old*)
	iNum_LenIgnHist_Old : USINT; (*Length of ignition events history [cycles] - Old*)
	iNum_IgnMiss_Max_Old : USINT; (*Maximum missing ignition events [cycles] - Old*)
	xTOF_OutputErr : TOF; (*Timer to disable W3545 during 3 s after and ITP change if KLS21 is active*)
	rCA_Ign_ActOld : ARRAY[0..24] OF REAL; (*Old ignition timing point*)
	bSA_ITP_Changed : BOOL; (*Ignition timing point changed*)
END_VAR
```

### Program Logical/SAFI/safi_pi (IEC, version 4.13.0) - + SAFI port injection

- safi_piCyclic.st (not readable text: treated as protected, skipped)

#### safi_pi.var
```iecst
(********************************************************************
 * COPYRIGHT -- INNIO
 ********************************************************************
 * Program: safi_pi
 * File: safi_pi.var
 * Author: weitzert
 * Created: February 23, 2010
 ********************************************************************
 * Local variables of program safi_pi
 ********************************************************************)
VAR
	bToggle : BOOL;
	usEventSum : UINT;
	bParaSendOK : BOOL;
	ucCylIndex : USINT;
	ucReDoCount : USINT;
	ucSAFIPIParaSend : USINT;
	SAFI_old : ARRAY[0..12] OF tSAFI;
	TON_PITest : TON;
	TON_TestDelay : TON;
	bToggle2 : BOOL;
	TON_SecondTick : TON;
	bAmmSeqClkP : BOOL;
	bHardwareErr : ARRAY[0..24] OF BOOL;
	AmmSeqHardwareErr : AmmSequence;
	bOpenErr : ARRAY[0..24] OF BOOL;
	bPIShutOff : ARRAY[0..24] OF BOOL;
	bIGNShutOff : ARRAY[0..24] OF BOOL;
	AmmSeqOpenErr : AmmSequence;
	AmmSeqPIShutOff : AmmSequence;
	AmmSeqIGNShutOff : AmmSequence;
	ucNrOfOpeningCyl : USINT;
	ucNrOfHwErr : USINT;
	bToggleEnab : BOOL;
	usCheckSum : UINT;
	bPIOpenCmd : BOOL;
	bPIOpenCmdOld : BOOL;
	bToggleOpen : BOOL;
	usCheckSum2 : UINT;
	ulDurAvgHelp : UDINT;
	usDurMaxHelp : UINT;
	usDurMinHelp : UINT;
	TON_AvgTick : TON;
	usFiFoLen : UINT;
	usCount : UINT;
	slCurrGradAvgHelp : DINT;
	ssCurrGradMaxHelp : INT;
	ssCurrGradMinHelp : INT;
	bPIDemagFail : ARRAY[0..24] OF BOOL;
	bPICurrCtrWarn : ARRAY[0..24] OF BOOL;
	bPICurrCtrRate : ARRAY[0..24] OF BOOL;
	bPISafLoopOpened : ARRAY[0..24] OF BOOL;
	AmmSeqPIDemagFail : AmmSequence;
	AmmSeqPICurrCtrWarn : AmmSequence;
	AmmSeqPICurrCtrRate : AmmSequence;
	TON_N_zero : TON;
	bSAFISendAllPIPara : BOOL;
	xTON_PICurGradFrozen : ARRAY[0..24] OF TON;
	xTON_PICurGradAltern : ARRAY[0..24] OF TON;
	iSA_PICurGrad_old1 : ARRAY[0..24] OF INT; (*PI close current gradient old value 1*)
	iSA_PICurGrad_old2 : ARRAY[0..24] OF INT; (*PI close current gradient old value 2*)
END_VAR
```

### Program Logical/SAFI/safi_kls (IEC, version 4.12.0) - + SAFI knock sensor

- safi_klsCyclic.st (not readable text: treated as protected, skipped)

- safi_klsInit.st (not readable text: treated as protected, skipped)

#### safi_kls.var
```iecst
VAR
	WMF4_D_Old : UINT;
	WMF4_B_Old : UINT;
	WMF3_D_Old : UINT;
	WMF3_B_Old : UINT;
	WMF2_D_Old : UINT;
	WMF2_B_Old : UINT;
	WMF1_D_Old : UINT;
	WMF1_B_Old : UINT;
	WMF_AD_Old : UINT;
	WMF_AB_Old : UINT;
	usMW_KLS3_Old : UINT;
	usMW_KLS2_Old : UINT;
	usMW_KLS1_Old : UINT;
	usEventSum : UINT;
	ucReDoCount : USINT;
	ucKLSMode_Old : ARRAY[0..12] OF USINT;
	ucCylIndex : USINT;
	ucCylinderCount : USINT;
	KLSGW4_Old : UINT;
	KLSGW3_Old : UINT;
	KLSGW2_Old : UINT;
	KLSGW1_Old : UINT;
	FenstF4_Old : USINT;
	FenstF3_Old : USINT;
	FenstF2_Old : USINT;
	FenstF1_Old : USINT;
	bToggle : BOOL;
	bParaSendOK : BOOL;
	AussSchwel_Old : UINT;
	TON_N_zero : TON;
	bSAFISendAllKLSPara : BOOL;
	ucSAFIKLSParaSend : USINT;
	iU_SAFI_Win1_old1 : ARRAY[0..24] OF INT;
	iU_SAFI_Win1_old2 : ARRAY[0..24] OF INT;
	xTON_Win1Frozen : ARRAY[0..24] OF TON;
	xTON_Win1Altern : ARRAY[0..24] OF TON;
	usMW_KLS4_Old : UINT; (*Average #kls__mdatas1 MUX 6/7 [cycles] - Old*)
	WMF5_B_Old : UINT; (* Start of window 5 [degCA] - Old*)
	WMF5_D_Old : UINT := 1; (* Duration of window  [degCA] - Old*)
	WMF6_B_Old : UINT; (* Start of window 6 [degCA] - Old*)
	WMF6_D_Old : UINT := 1; (* Duration of window 6 [degCA] - Old*)
	FenstF5_Old : USINT; (*Filter of KLS window 5 - Old*)
	FenstF6_Old : USINT; (*Filter of KLS window 6 - Old*)
	iNum_UpCurKlsSet_Old : USINT; (*KLS up curve settings - Old*)
END_VAR
```

### Program Logical/SAFI/safi_dmr (IEC, version 4.12.0) - + SAFI in-cylinder pressure sensor

- safi_dmrCyclic.st (not readable text: treated as protected, skipped)

- safi_dmrInit.st (not readable text: treated as protected, skipped)

#### safi_dmr.var
```iecst
VAR
	bToggle : BOOL;
	ssNEf_Old : INT;
	ssNEg_Old : INT;
	ucAussInt_Old : USINT;
	ucCylIndex : USINT;
	ucFuAU_Old : USINT;
	ucFuGZ_Old : USINT;
	ucFuIM_Old : USINT;
	ucUpCur_Old : ARRAY[0..12] OF USINT;
	ucFuNAE_Old : USINT;
	ucFuNE_Old : USINT;
	ucFuVL_Old : USINT;
	ucFuWE_Old : USINT;
	ucKuA_Old : USINT;
	ucReDoCount : USINT;
	ucSAFIEmpfCnt : USINT;
	usAussGW_Old : UINT;
	usEventSum : UINT;
	usGluehGW_Old : UINT;
	usIPEx_Old : UINT;
	usIPFa_Old : UINT;
	usIPGr_Old : UINT;
	usIPIt_Old : UINT;
	usIPKo_Old : UINT;
	usKlopfGW_Old : UINT;
	usMWEr_Old : UINT;
	usMWNGA_Old : UINT;
	usMWSt_Old : UINT;
	usNennDz_Old : UINT;
	usNETol_Old : UINT;
	usPolEx_Old : UINT;
	usthVW_Old : UINT;
	usVLFa_Old : UINT;
	usWMA_B_Old : UINT;
	usWMA_D_Old : UINT;
	usWMBB_B_Old : UINT;
	usWMBB_D_Old : UINT;
	usWMBD_B_Old : UINT;
	usWMBD_D_Old : UINT;
	usWMG_B_Old : UINT;
	usWMG_D_Old : UINT;
	usWMK_B_Old : UINT;
	usWMK_D_Old : UINT;
	usWMNEf_B_Old : UINT;
	usWMNEf_D_Old : UINT;
	usWMNEg_B_Old : UINT;
	usWMNEg_D_Old : UINT;
	usWMS_B_Old : UINT;
	usWMS_D_Old : UINT;
	usWMVL1_B_Old : UINT;
	usWMVL1_D_Old : UINT;
	usWMWE_B_Old : UINT;
	usWMWE_D_Old : UINT;
	bParaSendOK : BOOL;
	ssWEf_L_G_Old : INT;
	ssWEf_H_G_Old : INT;
	ucCylIndexN : USINT;
	usStartHP_Old : UINT;
	usDMRMode_Old : ARRAY[0..24] OF UINT;
	ucUP_Pos_Old : USINT;
	ssEmpf_Old : INT;
	ucCylCount : USINT;
	TON_N_zero : TON;
	bSAFISendAllDMRPara : BOOL;
	ucSAFIDMRParaSend : USINT;
	ssWEf_L_G : INT;
	ssWEf_H_G : INT;
	iPr_SAFI_Pmax : ARRAY[0..24] OF UINT; (*Pmax [10 mbar]*)
	iPr_SAFI_IMEP : ARRAY[0..24] OF UINT; (*IMEP [10 mbar]*)
	iPr_SAFI_Pmax_old1 : ARRAY[0..24] OF UINT; (*Pmax old value 1 [10 mbar]*)
	iPr_SAFI_Pmax_old2 : ARRAY[0..24] OF UINT; (*Pmax old value 2 [10 mbar]*)
	xTON_PmaxFrozen : ARRAY[0..24] OF TON;
	xTON_PmaxAltern : ARRAY[0..24] OF TON;
	iPr_SAFI_IMEP_old1 : ARRAY[0..24] OF UINT; (*IMEP old value 1 [10 mbar]*)
	iPr_SAFI_IMEP_old2 : ARRAY[0..24] OF UINT; (*IMEP old value 2 [10 mbar]*)
	xTON_IMEP_Frozen : ARRAY[0..24] OF TON;
	xTON_IMEP_Altern : ARRAY[0..24] OF TON;
END_VAR
```

### Program Logical/SAFI/safi_mpm (IEC, version 4.12.0) - + SAFI MPM control

- safi_mpmCyclic.st (not readable text: treated as protected, skipped)

#### safi_mpm.var - Local variables
```iecst
(********************************************************************
 * COPYRIGHT -- INNIO Company
 ********************************************************************
 * Program: safi_MPM
 * File: safi_MPM.var
 * Author: 105026877
 * Created: February 27, 2017
 ********************************************************************
 * Local variables of program safi_MPM
 ********************************************************************)
VAR
	TON_IgnPwr : TON;
	bMO_PwrRequest : BOOL;
	ucNrOfMPM : USINT;
	ucNrOfMPM_Req : USINT;
	bMO_PowerOverload : ARRAY[0..4] OF BOOL;
	bAmmSeqClkP : BOOL;
	AmmSeqIgnPowerOverload : AmmSequence;
	TON_SecondTick : TON;
	ucMpmCnt : USINT;
	TON_MO_PwrRequest : TON := (0);
	bOverloadCheck : BOOL := 0;
	bOverloadCheck2 : BOOL := 0;
	bOverloadCheck3 : BOOL := 0;
	bOverloadCheck4 : BOOL := 0;
	TON_IgnPwrOff : TON := (0);
	bMPM_Test : BOOL := 0;
	bMPM_StartOK : BOOL := 0;
	TON_FS_Overrule : TON := (0);
	ucNrOfMPM_ReqOld : USINT;
	bIgn_Dem_FS : BOOL; (*Ignition demand for FastStart*)
	TON_OverloadDelay : ARRAY[0..4] OF TON;
END_VAR
```

### Program Logical/SAFI/safi_vcd (IEC, version 4.13.0) - + SAFI valve closure detection

- safi_vcdCyclic.st (not readable text: treated as protected, skipped)

- safi_vcdInit.st (not readable text: treated as protected, skipped)

#### safi_vcd.var - Local variables
```iecst
(********************************************************************
 * COPYRIGHT -- INNIO
 ********************************************************************
 * Program: safi_vcd
 * File: safi_vcd.var
 * Author: 212567725
 * Created: December 18, 2018
 ********************************************************************
 * Local variables of program safi_vcd
 ********************************************************************)
VAR
	ucCylinderCount : USINT;
	ucCylIndex : USINT;
	SAFI_EVCD : ARRAY[0..24] OF fSAFI_VCD; (*Function processing the EVC timing*)
	rNum_VCD_StdLim : REAL;
	SAFI_IVCD : ARRAY[0..24] OF fSAFI_VCD; (*Function processing the IVC timing*)
	bWin3High : ARRAY[0..24] OF BOOL; (*Error bit: EVC noise too high*)
	bWin4High : ARRAY[0..24] OF BOOL; (*Error bit: IVC noise too high*)
	iCA_Win3Avg : UINT; (*EVC timing average of all cylinders*)
	iCA_Win3AvgSum : UDINT;
	iCA_Win3Max : UINT; (*EVC timing maximum of all cylinders*)
	iCA_Win3Min : UINT; (*EVC timing minimum of all cylinders*)
	iCA_Win3_timing : ARRAY[0..24] OF UINT; (*EVC timing signal from SAFI*)
	iCA_Win4Avg : UINT; (*IVC timing average of all cylinders*)
	iCA_Win4AvgSum : UDINT;
	iCA_Win4Max : UINT; (*IVC timing maximum of all cylinders*)
	iCA_Win4Min : UINT; (*IVC timing minimum of all cylinders*)
	iCA_Win4_timing : ARRAY[0..24] OF UINT; (*IVC timing signal from SAFI*)
	iCnt_Win3 : USINT;
	iCnt_Win3LimitCount : ARRAY[0..24] OF USINT;
	iCnt_Win4 : USINT;
	iCnt_Win4LimitCount : ARRAY[0..24] OF USINT;
	iU_Win3Avg : UINT; (*EVC noise average of all cylinders*)
	iU_Win3AvgSum : UDINT;
	iU_Win3Max : UINT; (*EVC noise maximum of all cylinders*)
	iU_Win3Min : UINT; (*EVC noise minimum of all cylinders*)
	iU_Win3_noise : ARRAY[0..24] OF UINT; (*EVC noise signal from SAFI*)
	iU_Win4Avg : UINT; (*IVC noise average of all cylinders*)
	iU_Win4AvgSum : UDINT;
	iU_Win4Max : UINT; (*IVC noise maximum of all cylinders*)
	iU_Win4Min : UINT; (*IVC noise minimum of all cylinders*)
	iU_Win4_noise : ARRAY[0..24] OF UINT; (*IVC noise signal from SAFI*)
	bAmmSeqClkP : BOOL;
	AmmSeqInValveErr : AmmSequence;
	AmmSeqExValveErr : AmmSequence;
	TON_SecondTick : TON;
	xTON_ValveLashSet : ARRAY[0..24] OF TON; (*2 minutes delay to reset the "Valve lash adjusted" tick boxes*)
	xTON_ValveLashSetAll : TON; (*2 minutes delay to reset the "Valve lash adjusted" tick boxes*)
	iNum_PeakPercLim : UINT; (*Limit in pecentage of occurences of the 2nd highest peak*)
	AmmSeqExValveUnb : AmmSequence;
	AmmSeqInValveUnb : AmmSequence;
	b_EVC_Unb : ARRAY[0..24] OF BOOL; (*Valve unbalance detected - Exhaust*)
	b_IVC_Unb : ARRAY[0..24] OF BOOL; (*Valve unbalance detected - Intake*)
	iU_EVCNoiseLimit : UINT; (*EVC noise maximum limit*)
	iU_IVCNoiseLimit : UINT; (*IVC noise maximum limit*)
	xTP_DelayStart : TP; (*Timer TRUE for 20 minutes after engine start*)
	iCnt_CAWin3 : USINT;
	iCnt_CAWin4 : USINT;
END_VAR
```

### Program Logical/SAFI/IN_SA (IEC, version 4.12.0) - + SAFI IN task

- IN_SACyclic.st (not readable text: treated as protected, skipped)

### Program Logical/SAFI/CurveUpL (IEC, version 4.07.0) - + SAFI curve upload

- CurveUpLCyclic.st (not readable text: treated as protected, skipped)

- CurveUpLInit.st (not readable text: treated as protected, skipped)

#### CurveUpL.var - Local variables
```iecst
(********************************************************************
 * COPYRIGHT -- INNIO Company
 ********************************************************************
 * Program: UpLoadCurve
 * File: UpLoadCurve.var
 * Author: 120011115
 * Created: April 23, 2013
 ********************************************************************
 * Local variables of program UpLoadCurve
 ********************************************************************)
VAR
	tRealTime : rtctime_typ; (* time structure *)
	DTGetTime_RPS : DTGetTime;
	bActive : ARRAY[0..12] OF BOOL;
	bActiveCounter : ARRAY[0..12] OF UINT;
	bAllHigh : BOOL;
	bCANMiss : BOOL;
	bCANWait : BOOL;
	bCreateDataObj : BOOL;
	bErrPermSlowDown : BOOL;
	bReleaseH : ARRAY[0..12] OF BOOL;
	bReleaseL : ARRAY[0..12] OF BOOL;
	bWriteDataObj : BOOL;
	CA_old_H : UINT;
	CA_old_L : UINT;
	DatObjCreate_01 : DatObjCreate;
	DatObjDelete_PermMem : DatObjDelete;
	DatObjInfo_01 : DatObjInfo;
	DatObjRead_01 : DatObjRead;
	DatObjWrite_01 : DatObjWrite;
	EngineStop : BOOL;
	Error_H_New : ARRAY[0..12] OF BOOL;
	Error_H_Old : ARRAY[0..12] OF BOOL;
	Error_L_New : ARRAY[0..12] OF BOOL;
	Error_L_Old : ARRAY[0..12] OF BOOL;
	iCycleCounter : UINT;
	IdCyl : USINT;
	iDelayCounter : UINT;
	IdSAFI : USINT;
	idx : USINT;
	ManCount : USINT;
	ModulName : STRING[35]; (*Bugfix V4.07*)
	N_Cycles : UINT;
	perm_vers : UINT;
	pm_Cup : tCup_Pm;
	pm_Error : UINT;
	pm_id : UDINT;
	pm_len : UDINT;
	pm_p : UDINT;
	TON_WarnDelay : TON;
	TON_WritePMEM : TON;
	uCountMissH : USINT;
	uCountMissL : USINT;
	ulChecksum : UDINT;
	ulChecksumOld : UDINT;
	ulChkValue : UDINT;
	ulPMPointer : UDINT;
	usPress : ARRAY[0..12] OF Pressure;
	write_once : BOOL;
	xTON_01 : TON;
	ucSAFI_ID : USINT;
	i : UINT;
END_VAR
VAR CONSTANT
	ERR_NOERROR : UINT := 0;
END_VAR
VAR
	bBlock_MinFileAge : BOOL := FALSE; (*V4.07*)
	TON_BlockMinFileAge : TON; (*V4.07*)
	iPM_WriteCnt : UDINT; (*V4.07*)
END_VAR
```

### Program Logical/SAFI/OUT_SA (IEC, version 4.11.0) - + SAFI OUT task

- OUT_SACyclic.st (not readable text: treated as protected, skipped)

### Program Logical/SAFI/ParSA (IEC, version 4.06.0) - + SAFI Parameter

- perm_par.st (not readable text: treated as protected, skipped)

#### perm_par.var
```iecst
VAR
	tParaIntern : ParaHandler_typ; (*Connector type to perm_par*)
	tMM2ParaBase_ReadBack : MM2ParaBase_type; (*INTERNAL! V4.06 new readback structure for information from previous tasks*)
	bWriteDataObj : BOOL; (* TRUE=write data object module *)
	bDataObjLenErr : BOOL; (*Error occured in permem: data module size missmatch*)
	bCreateDataObj : BOOL; (* TRUE=create new data object *)
	bWriteOnce : BOOL; (* write permanent memory once *)
	DatObjCreate_01 : DatObjCreate; (* data object create *)
	DatObjInfoBak_02 : DatObjInfo; (* data object info *)
	DatObjDelete_01 : DatObjDelete; (* data object delete *)
	DatObjRead_01 : DatObjRead; (* data object read *)
	DatObjRead_02 : DatObjRead; (* manual initiated data object read *)
	DatObjWrite_01 : DatObjWrite; (* data object write *)
	DatObjDelete_02 : DatObjDelete; (* data object delete *)
	DatObjDelete_11 : DatObjDelete; (*Delete Backup File*)
	DatObjInfo_01 : DatObjInfo; (* data object info *)
	DatObjInfo_02 : DatObjInfo; (* data object info *)
	szModuleName : STRING[35]; (* module name of object *)
	szModuleNameBackup : STRING[35]; (* module name of posiibly created backup object *)
	DatObjCopy_01 : DatObjCopy;
	bCopyDataObj : BOOL;
	TON_WarnDelay : TON;
	TON_WritePMEM : TON; (* delay write permanent memory *)
	ulPMPointer : UDINT; (* adress of actual checksum value *)
	ulChecksum : UDINT; (* parameter checksum value *)
	pm_len : UDINT; (* permanent value lenght *)
	ulChecksumOld : UDINT; (* last vlaue of parameter checksum *)
	ulChkValue : UDINT; (* actual value of parameter pointer *)
	pm_id : UDINT; (* permanent value identifier *)
	pm_p : UDINT; (* permanent value pointer *)
	DatObjInfo_META : DatObjInfo;
	DatObjRead_META : DatObjRead;
	szMetaDataRaw : STRING[2000];
	szMetaData : ARRAY[0..4] OF STRING[35];
	szMetaDataVis : ARRAY[0..3] OF STRING[35];
	ssIndex : INT;
	ssCount : INT;
	ucMetaDataRaw : ARRAY[0..2000] OF USINT;
	ssCount2 : INT;
	szMetaDataFile : STRING[10];
	szText1 : STRING[20];
	pv_adr_IN_XX_tPB2MM : UDINT;
	pv_lng : UDINT;
	pv_lng_IN_XX_tPB2MM : UDINT;
	pv_lng_OUT_XX_tPB2MM : UDINT;
	szText2 : STRING[20];
	pv_adr_OUT_XX_tXX2PB : UDINT;
END_VAR
VAR CONSTANT
	ERR_NOERROR : UINT := 0;
END_VAR
VAR
	usPMWriteCnt : UINT;
	pm_Error : UDINT; (* permanent value error *) (* Deleted: pm : ParaMem_typ; permanent memory tags mathias, 22.8.11*)
	fun_Error : UDINT := 0; (*state > 0 = function error*)
	xLocalParaCheck : ParaCheckFUB; (*local function instance to check parameter values*)
	TON_ParaSetupOk : TON;
	bParaCheckSystemOk : BOOL;
	iDebug_ParaOkChecked : UDINT;
	bRestoreBackupDataObj : BOOL := FALSE;
	bRestoreDataObjContent : BOOL := FALSE;
	pm_id_backup : UDINT;
	pm_p_Backup : UDINT;
	DatObjCopy_02 : DatObjCopy;
	bDeleteBackupDataObj : BOOL := FALSE; (*Command to delete backup data module file on purpose*)
	bDebugPara : ARRAY[0..5] OF BOOL;
	ssIndex2 : INT;
	ssIndex3 : INT;
	ssIndex4 : INT;
	ssIndexVis : INT;
	szText : STRING[40];
	pv_adr_Para : UDINT;
	szParaSnippet : ARRAY[0..5] OF STRING[150];
	szParaIndex : STRING[10];
	slValue : DINT;
	iModuleDLD_ResetCount : INT;
	bDownloadDetected : BOOL;
	bFlagParaStructCopyWorking : BOOL; (*true, if cyclic para copying is active, 1 false cycle at every copy *)
	bStoreInitParaInDataObj : BOOL := FALSE;
	bTestflag : BOOL;
	bReadOutMETA_Once : BOOL;
	tParaCheck_iPvAdress : ARRAY[0..5] OF UDINT;
	tParaCheck_iPvLengt : ARRAY[0..5] OF UDINT;
	tParaCheck_rPvValue : ARRAY[0..5] OF REAL;
	tParaCheck_rRangeMIN : ARRAY[0..5] OF REAL;
	tParaCheck_rRangeMAX : ARRAY[0..5] OF REAL;
	tParaCheck_szPvName : ARRAY[0..5] OF STRING[35];
	ssFormatDetected : INT;
	szMetaDataPart : STRING[150];
	szFullTaskName : STRING[35];
	szFullMetaModuleName : STRING[35];
	debugLen : INT;
	debugSize : INT := 0;
	strcat_adr1 : UDINT;
	strcat_adr2 : UDINT;
	ssIndexTN : INT;
	bAlternate : BOOL;
	n : INT;
	iAlternateChecksum : DINT;
	iAlternateChecksumOld : DINT;
	ulDebugChkValue : ARRAY[0..999] OF UDINT;
	Adr1 : UDINT;
	Adr2 : UDINT;
	usPMWriteCntStepsize : UINT := 1; (*different step sizes to help debug*)
	usPMWriteCntXOR : UINT;
	usPMWriteCntAltSum : UINT;
	ulAdrPM : UDINT;
	usChkValuePM : USINT;
	ulAdrPara : UDINT;
	ulPara_len : UDINT;
	usChkValuePara : USINT;
	iDebugCountPMDifferences : DINT := 0;
	bEngineRunDetected : BOOL; (*detection status bit autocommand 100 /101  for engine run state*)
	ucMetaDataDebugInfoLine : ARRAY[0..24] OF STRING[80];
	ssIndexMand : INT := 0;
	szMetaDataMand : STRING[35];
	iMyErrorInfo_Autoreset : DINT; (*internal autoreset counter*)
	ssIndex_Version : INT; (*internal*)
	ssIndex_BU : INT; (*internal*)
	ssIndex_BU2 : INT; (*internal*)
END_VAR
```

### Program Logical/SAFI/MsgSA (IEC, version 4.14.0) - + SAFI Messages

- MsgSACyclic.st (not readable text: treated as protected, skipped)

- MsgSAInit.st (not readable text: treated as protected, skipped)
